KUKA KRL program: Station400_IMM.src, Station400_IMM.dat

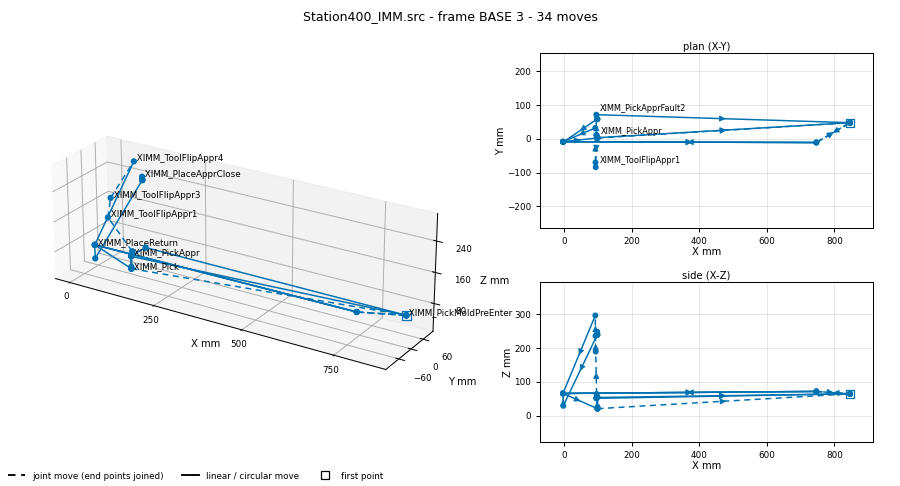
[picture p0: tool path of Station400_IMM.src in frame BASE 3, 34 of 42 moves have a stored position in this frame; points joined in program order, loops and branches not executed]
--- Station400_IMM.src ---
&ACCESS RVO1
&REL 170
&PARAM DISKPATH = KRC:\R1\Program
DEF Station400_IMM()
   ;FOLD INI;%{PE}
      ;FOLD BASISTECH INI
         GLOBAL INTERRUPT DECL 3 WHEN $STOPMESS == TRUE DO IR_STOPM()
         INTERRUPT ON 3
         BAS(#INITMOV, 0)
      ;ENDFOLD (BASISTECH INI)
      ;FOLD USER INI
         ;Make your modifications here
      ;ENDFOLD (USER INI)
      ;ENDFOLD (INI)
 RetryEntry:
 RtoIMM_MoldOpenEnable=True
 RtoPLC_FinishGripClose=False
 RtoPLC_FinishGripOpen=True
 wait sec .25
 RtoPLC_FinishGripOpen=False
 RobotCell_Error=False


;FOLD SPTP IMM_A1turn Vel=100 % PDAT4 Tool[0] Base[0] ;%{PE}
;FOLD Parameters ;%{h}
;Params IlfProvider=kukaroboter.basistech.inlineforms.movement.spline; Kuka.IsGlobalPoint=False; Kuka.PointName=IMM_A1turn; Kuka.BlendingEnabled=False; Kuka.MoveDataPtpName=PDAT4; Kuka.VelocityPtp=100; Kuka.VelocityFieldEnabled=True; Kuka.ColDetectFieldEnabled=True; Kuka.CurrentCDSetIndex=0; Kuka.MovementParameterFieldEnabled=True; IlfCommand=SPTP
;ENDFOLD
SPTP XIMM_A1turn WITH $VEL_AXIS[1] = SVEL_JOINT(100.0), $TOOL = STOOL2(FIMM_A1turn), $BASE = SBASE(FIMM_A1turn.BASE_NO), $IPO_MODE = SIPO_MODE(FIMM_A1turn.IPO_FRAME), $LOAD = SLOAD(FIMM_A1turn.TOOL_NO), $ACC_AXIS[1] = SACC_JOINT(PPDAT4), $APO = SAPO_PTP(PPDAT4), $GEAR_JERK[1] = SGEAR_JERK(PPDAT4), $COLLMON_TOL_PRO[1] = USE_CM_PRO_VALUES(0)
;ENDFOLD

Wait For IMMtoR_OpEnable==True
 Wait For RtoIMM_RobotWithIMM==False


;FOLD Wait for ejector backward signals,
$TIMER_STOP[2]=True ;stop timer
$TIMER[2]=0 ;reset timer
$TIMER_STOP[2]=False ;stop timer
Loop
       If $TIMER[2]>=5000 Then
              $TIMER_STOP[2]=True ;stop timer
              $TIMER[2]=0 ;reset timer
              IMMtoR_PreEntrErrorEjBck=True
              wait sec 0.25
              IMMtoR_PreEntrErrorEjBck=False
              Wait For IMMtoR_OpEnable==False
              GOTO RetryEntry
       EndIf
       If IMMtoR_EjectPosBck==True Then
              Exit
       EndIf
EndLoop
 ;ENDFOLD

;FOLD Wait for mold open signal, fault after 10 seconds of waiting, then move in over sprue, down and into mold pick position, turn on suction cups
$TIMER_STOP[2]=True ;stop timer
$TIMER[2]=0 ;reset timer
$TIMER_STOP[2]=False ;stop timer

Loop

       If $TIMER[2]>=5000 Then
              $TIMER_STOP[2]=True ;stop timer
              $TIMER[2]=0 ;reset timer
              IMMtoR_PlaceErrorMoldOpn=True
              wait sec 0.5
              IMMtoR_PlaceErrorMoldOpn=False
              Wait For IMMtoR_OpEnable==False
              GOTO RetryEntry
       EndIF

       If ((IMMtoR_MoldOpen==True) AND ((IMMtoR_PartInjected==True) Or (RtoIMM_SeqNumber<>0)))  Then
              If IMMtoR_Rejected==True Then
                     RtoPLC_ToolFinReject=True
              EndIf
              RtoIMM_MoldCloseEnable=False
              RtoIMM_MoldAreaFree=False
   ;FOLD SPTP IMM_PickMoldPreEnter CONT Vel=100 % PDAT1 Tool[2]:FinishedPlace Base[3]:IMM ;%{PE}
      ;FOLD Parameters ;%{h}
         ;Params IlfProvider=kukaroboter.basistech.inlineforms.movement.spline; Kuka.IsGlobalPoint=False; Kuka.PointName=IMM_PickMoldPreEnter; Kuka.BlendingEnabled=True; Kuka.MoveDataPtpName=PDAT1; Kuka.VelocityPtp=100; Kuka.VelocityFieldEnabled=True; Kuka.ColDetectFieldEnabled=True; Kuka.CurrentCDSetIndex=0; Kuka.MovementParameterFieldEnabled=True; IlfCommand=SPTP
      ;ENDFOLD
      SPTP XIMM_PickMoldPreEnter WITH $VEL_AXIS[1] = SVEL_JOINT(100.0), $TOOL = STOOL2(FIMM_PickMoldPreEnter), $BASE = SBASE(FIMM_PickMoldPreEnter.BASE_NO), $IPO_MODE = SIPO_MODE(FIMM_PickMoldPreEnter.IPO_FRAME), $LOAD = SLOAD(FIMM_PickMoldPreEnter.TOOL_NO), $ACC_AXIS[1] = SACC_JOINT(PPDAT1), $APO = SAPO_PTP(PPDAT1), $GEAR_JERK[1] = SGEAR_JERK(PPDAT1), $COLLMON_TOL_PRO[1] = USE_CM_PRO_VALUES(0) C_Spl
      ;ENDFOLD
;FOLD SLIN IMM_PickApprOvrSpru CONT Vel=1.5 m/s CPDAT01 Tool[1]:BlankPick Base[4]:SprueCutter ;%{PE}
;FOLD Parameters ;%{h}
;Params IlfProvider=kukaroboter.basistech.inlineforms.movement.spline; Kuka.IsGlobalPoint=False; Kuka.PointName=IMM_PickApprOvrSpru; Kuka.BlendingEnabled=True; Kuka.MoveDataName=CPDAT01; Kuka.VelocityPath=1.5; Kuka.VelocityFieldEnabled=True; Kuka.ColDetectFieldEnabled=True; Kuka.CurrentCDSetIndex=0; Kuka.MovementParameterFieldEnabled=True; IlfCommand=SLIN
;ENDFOLD
SLIN XIMM_PickApprOvrSpru WITH $VEL = SVEL_CP(1.5, , LCPDAT01), $TOOL = STOOL2(FIMM_PickApprOvrSpru), $BASE = SBASE(FIMM_PickApprOvrSpru.BASE_NO), $IPO_MODE = SIPO_MODE(FIMM_PickApprOvrSpru.IPO_FRAME), $LOAD = SLOAD(FIMM_PickApprOvrSpru.TOOL_NO), $ACC = SACC_CP(LCPDAT01), $ORI_TYPE = SORI_TYP(LCPDAT01), $APO = SAPO(LCPDAT01), $JERK = SJERK(LCPDAT01), $COLLMON_TOL_PRO[1] = USE_CM_PRO_VALUES(0) C_Spl
;ENDFOLD
;FOLD SLIN IMM_PickAppr Vel=1 m/s CPDAT2 Tool[2]:FinishedPlace Base[3]:IMM ;%{PE}
;FOLD Parameters ;%{h}
;Params IlfProvider=kukaroboter.basistech.inlineforms.movement.spline; Kuka.IsGlobalPoint=False; Kuka.PointName=IMM_PickAppr; Kuka.BlendingEnabled=False; Kuka.MoveDataName=CPDAT2; Kuka.VelocityPath=1; Kuka.VelocityFieldEnabled=True; Kuka.ColDetectFieldEnabled=True; Kuka.CurrentCDSetIndex=0; Kuka.MovementParameterFieldEnabled=True; IlfCommand=SLIN
;ENDFOLD
SLIN XIMM_PickAppr WITH $VEL = SVEL_CP(1.0, , LCPDAT2), $TOOL = STOOL2(FIMM_PickAppr), $BASE = SBASE(FIMM_PickAppr.BASE_NO), $IPO_MODE = SIPO_MODE(FIMM_PickAppr.IPO_FRAME), $LOAD = SLOAD(FIMM_PickAppr.TOOL_NO), $ACC = SACC_CP(LCPDAT2), $ORI_TYPE = SORI_TYP(LCPDAT2), $APO = SAPO(LCPDAT2), $JERK = SJERK(LCPDAT2), $COLLMON_TOL_PRO[1] = USE_CM_PRO_VALUES(0)
;ENDFOLD
;FOLD SLIN IMM_Pick Vel=0.05 m/s CPDAT1 Tool[2]:FinishedPlace Base[3]:IMM ;%{PE}
;FOLD Parameters ;%{h}
;Params IlfProvider=kukaroboter.basistech.inlineforms.movement.spline; Kuka.IsGlobalPoint=False; Kuka.PointName=IMM_Pick; Kuka.BlendingEnabled=False; Kuka.MoveDataName=CPDAT1; Kuka.VelocityPath=0.05; Kuka.VelocityFieldEnabled=True; Kuka.ColDetectFieldEnabled=True; Kuka.CurrentCDSetIndex=0; Kuka.MovementParameterFieldEnabled=True; IlfCommand=SLIN
;ENDFOLD
SLIN XIMM_Pick WITH $VEL = SVEL_CP(0.05, , LCPDAT1), $TOOL = STOOL2(FIMM_Pick), $BASE = SBASE(FIMM_Pick.BASE_NO), $IPO_MODE = SIPO_MODE(FIMM_Pick.IPO_FRAME), $LOAD = SLOAD(FIMM_Pick.TOOL_NO), $ACC = SACC_CP(LCPDAT1), $ORI_TYPE = SORI_TYP(LCPDAT1), $APO = SAPO(LCPDAT1), $JERK = SJERK(LCPDAT1), $COLLMON_TOL_PRO[1] = USE_CM_PRO_VALUES(0)
;ENDFOLD
              RtoPLC_FinishCupAVac=True
              RtoPLC_FinishCupBVac=True
              $TIMER_STOP[2]=True ;stop timer
              $TIMER[2]=0 ;reset timer
              Exit
       EndIf

       If ((IMMtoR_MoldOpen==True) AND ((IMMtoR_PartInjected==False) And (RtoIMM_SeqNumber==0)))  Then
              RtoIMM_MoldCloseEnable=False
              RtoIMM_MoldAreaFree=False
   ;FOLD SPTP IMM_PickMoldPreEnter CONT Vel=100 % PDAT1 Tool[2]:FinishedPlace Base[3]:IMM ;%{PE}
      ;FOLD Parameters ;%{h}
         ;Params IlfProvider=kukaroboter.basistech.inlineforms.movement.spline; Kuka.IsGlobalPoint=False; Kuka.PointName=IMM_PickMoldPreEnter; Kuka.BlendingEnabled=True; Kuka.MoveDataPtpName=PDAT1; Kuka.VelocityPtp=100; Kuka.VelocityFieldEnabled=True; Kuka.ColDetectFieldEnabled=True; Kuka.CurrentCDSetIndex=0; Kuka.MovementParameterFieldEnabled=True; IlfCommand=SPTP
      ;ENDFOLD
      SPTP XIMM_PickMoldPreEnter WITH $VEL_AXIS[1] = SVEL_JOINT(100.0), $TOOL = STOOL2(FIMM_PickMoldPreEnter), $BASE = SBASE(FIMM_PickMoldPreEnter.BASE_NO), $IPO_MODE = SIPO_MODE(FIMM_PickMoldPreEnter.IPO_FRAME), $LOAD = SLOAD(FIMM_PickMoldPreEnter.TOOL_NO), $ACC_AXIS[1] = SACC_JOINT(PPDAT1), $APO = SAPO_PTP(PPDAT1), $GEAR_JERK[1] = SGEAR_JERK(PPDAT1), $COLLMON_TOL_PRO[1] = USE_CM_PRO_VALUES(0) C_Spl
      ;ENDFOLD
;FOLD SPTP IMM_PlaceMoldReturn Vel=100 % PDAT15 Tool[1]:BlankPick Base[3]:IMM ;%{PE}
;FOLD Parameters ;%{h}
;Params IlfProvider=kukaroboter.basistech.inlineforms.movement.spline; Kuka.IsGlobalPoint=False; Kuka.PointName=IMM_PlaceMoldReturn; Kuka.BlendingEnabled=False; Kuka.MoveDataPtpName=PDAT15; Kuka.VelocityPtp=100; Kuka.VelocityFieldEnabled=True; Kuka.ColDetectFieldEnabled=True; Kuka.CurrentCDSetIndex=0; Kuka.MovementParameterFieldEnabled=True; IlfCommand=SPTP
;ENDFOLD
SPTP XIMM_PlaceMoldReturn WITH $VEL_AXIS[1] = SVEL_JOINT(100.0), $TOOL = STOOL2(FIMM_PlaceMoldReturn), $BASE = SBASE(FIMM_PlaceMoldReturn.BASE_NO), $IPO_MODE = SIPO_MODE(FIMM_PlaceMoldReturn.IPO_FRAME), $LOAD = SLOAD(FIMM_PlaceMoldReturn.TOOL_NO), $ACC_AXIS[1] = SACC_JOINT(PPDAT15), $APO = SAPO_PTP(PPDAT15), $GEAR_JERK[1] = SGEAR_JERK(PPDAT15), $COLLMON_TOL_PRO[1] = USE_CM_PRO_VALUES(0)
;ENDFOLD

;FOLD SLIN IMM_PlaceReturn Vel=2 m/s CPDAT23 Tool[1]:BlankPick Base[3]:IMM ;%{PE}
;FOLD Parameters ;%{h}
;Params IlfProvider=kukaroboter.basistech.inlineforms.movement.spline; Kuka.IsGlobalPoint=False; Kuka.PointName=IMM_PlaceReturn; Kuka.BlendingEnabled=False; Kuka.MoveDataName=CPDAT23; Kuka.VelocityPath=2; Kuka.VelocityFieldEnabled=True; Kuka.ColDetectFieldEnabled=True; Kuka.CurrentCDSetIndex=0; Kuka.MovementParameterFieldEnabled=True; IlfCommand=SLIN
;ENDFOLD
SLIN XIMM_PlaceReturn WITH $VEL = SVEL_CP(2.0, , LCPDAT23), $TOOL = STOOL2(FIMM_PlaceReturn), $BASE = SBASE(FIMM_PlaceReturn.BASE_NO), $IPO_MODE = SIPO_MODE(FIMM_PlaceReturn.IPO_FRAME), $LOAD = SLOAD(FIMM_PlaceReturn.TOOL_NO), $ACC = SACC_CP(LCPDAT23), $ORI_TYPE = SORI_TYP(LCPDAT23), $APO = SAPO(LCPDAT23), $JERK = SJERK(LCPDAT23), $COLLMON_TOL_PRO[1] = USE_CM_PRO_VALUES(0)
;ENDFOLD
              $TIMER_STOP[2]=True ;stop timer
              $TIMER[2]=0 ;reset timer
              GoTo PlaceInMold
       EndIf
EndLoop
;ENDFOLD

;FOLD Wait for suction cup vacuum signals, fault after 10 seconds of waiting (and back out of mold), move ejector forward,
$TIMER_STOP[2]=True ;stop timer
$TIMER[2]=0 ;reset timer
$TIMER_STOP[2]=False ;stop timer
Loop

       If $TIMER[2]>=5000 Then
              $TIMER_STOP[2]=True ;stop timer
              $TIMER[2]=0 ;reset timer
              If PLCtoR_FinishCupAVacOn==False Then
                     RtoIMM_PickErrorVG528=True

              EndIf
              If PLCtoR_FinishCupBVacOn==False Then
                     RtoIMM_PickErrorVG530=True

              EndIf
              Wait Sec .15
              RtoPLC_FinishCupAVac=False
              RtoPLC_FinishCupBVac=False
              RtoPLC_FinishCupABlow=True
              RtoPLC_FinishCupBBlow=True
              Wait Sec .15
              RtoPLC_FinishCupABlow=False
              RtoPLC_FinishCupBBlow=False
              RtoIMM_PickErrorVG528=False
              RtoIMM_PickErrorVG530=False
              Wait For IMMtoR_OpEnable==False
              $OV_PRO=30
              ;FOLD SLIN IMM_Pick Vel=0.05 m/s CPDAT1 Tool[2]:FinishedPlace Base[3]:IMM ;%{PE}
;FOLD Parameters ;%{h}
;Params IlfProvider=kukaroboter.basistech.inlineforms.movement.spline; Kuka.IsGlobalPoint=False; Kuka.PointName=IMM_Pick; Kuka.BlendingEnabled=False; Kuka.MoveDataName=CPDAT1; Kuka.VelocityPath=0.05; Kuka.VelocityFieldEnabled=True; Kuka.ColDetectFieldEnabled=True; Kuka.CurrentCDSetIndex=0; Kuka.MovementParameterFieldEnabled=True; IlfCommand=SLIN
;ENDFOLD
SLIN XIMM_Pick WITH $VEL = SVEL_CP(0.05, , LCPDAT1), $TOOL = STOOL2(FIMM_Pick), $BASE = SBASE(FIMM_Pick.BASE_NO), $IPO_MODE = SIPO_MODE(FIMM_Pick.IPO_FRAME), $LOAD = SLOAD(FIMM_Pick.TOOL_NO), $ACC = SACC_CP(LCPDAT1), $ORI_TYPE = SORI_TYP(LCPDAT1), $APO = SAPO(LCPDAT1), $JERK = SJERK(LCPDAT1), $COLLMON_TOL_PRO[1] = USE_CM_PRO_VALUES(0)
;ENDFOLD
;FOLD SLIN IMM_PickAppr Vel=1 m/s CPDAT2 Tool[2]:FinishedPlace Base[3]:IMM ;%{PE}
;FOLD Parameters ;%{h}
;Params IlfProvider=kukaroboter.basistech.inlineforms.movement.spline; Kuka.IsGlobalPoint=False; Kuka.PointName=IMM_PickAppr; Kuka.BlendingEnabled=False; Kuka.MoveDataName=CPDAT2; Kuka.VelocityPath=1; Kuka.VelocityFieldEnabled=True; Kuka.ColDetectFieldEnabled=True; Kuka.CurrentCDSetIndex=0; Kuka.MovementParameterFieldEnabled=True; IlfCommand=SLIN
;ENDFOLD
SLIN XIMM_PickAppr WITH $VEL = SVEL_CP(1.0, , LCPDAT2), $TOOL = STOOL2(FIMM_PickAppr), $BASE = SBASE(FIMM_PickAppr.BASE_NO), $IPO_MODE = SIPO_MODE(FIMM_PickAppr.IPO_FRAME), $LOAD = SLOAD(FIMM_PickAppr.TOOL_NO), $ACC = SACC_CP(LCPDAT2), $ORI_TYPE = SORI_TYP(LCPDAT2), $APO = SAPO(LCPDAT2), $JERK = SJERK(LCPDAT2), $COLLMON_TOL_PRO[1] = USE_CM_PRO_VALUES(0)
;ENDFOLD
;FOLD SLIN IMM_PickApprOvrSpru CONT Vel=1.5 m/s CPDAT01 Tool[1]:BlankPick Base[4]:SprueCutter ;%{PE}
;FOLD Parameters ;%{h}
;Params IlfProvider=kukaroboter.basistech.inlineforms.movement.spline; Kuka.IsGlobalPoint=False; Kuka.PointName=IMM_PickApprOvrSpru; Kuka.BlendingEnabled=True; Kuka.MoveDataName=CPDAT01; Kuka.VelocityPath=1.5; Kuka.VelocityFieldEnabled=True; Kuka.ColDetectFieldEnabled=True; Kuka.CurrentCDSetIndex=0; Kuka.MovementParameterFieldEnabled=True; IlfCommand=SLIN
;ENDFOLD
SLIN XIMM_PickApprOvrSpru WITH $VEL = SVEL_CP(1.5, , LCPDAT01), $TOOL = STOOL2(FIMM_PickApprOvrSpru), $BASE = SBASE(FIMM_PickApprOvrSpru.BASE_NO), $IPO_MODE = SIPO_MODE(FIMM_PickApprOvrSpru.IPO_FRAME), $LOAD = SLOAD(FIMM_PickApprOvrSpru.TOOL_NO), $ACC = SACC_CP(LCPDAT01), $ORI_TYPE = SORI_TYP(LCPDAT01), $APO = SAPO(LCPDAT01), $JERK = SJERK(LCPDAT01), $COLLMON_TOL_PRO[1] = USE_CM_PRO_VALUES(0) C_Spl
;ENDFOLD
;FOLD SLIN IMM_PickMoldPreEnter Vel=2 m/s CPDAT29 Tool[2]:FinishedPlace Base[3]:IMM ;%{PE}
;FOLD Parameters ;%{h}
;Params IlfProvider=kukaroboter.basistech.inlineforms.movement.spline; Kuka.IsGlobalPoint=False; Kuka.PointName=IMM_PickMoldPreEnter; Kuka.BlendingEnabled=False; Kuka.MoveDataName=CPDAT29; Kuka.VelocityPath=2; Kuka.VelocityFieldEnabled=True; Kuka.ColDetectFieldEnabled=True; Kuka.CurrentCDSetIndex=0; Kuka.MovementParameterFieldEnabled=True; IlfCommand=SLIN
;ENDFOLD
SLIN XIMM_PickMoldPreEnter WITH $VEL = SVEL_CP(2.0, , LCPDAT29), $TOOL = STOOL2(FIMM_PickMoldPreEnter), $BASE = SBASE(FIMM_PickMoldPreEnter.BASE_NO), $IPO_MODE = SIPO_MODE(FIMM_PickMoldPreEnter.IPO_FRAME), $LOAD = SLOAD(FIMM_PickMoldPreEnter.TOOL_NO), $ACC = SACC_CP(LCPDAT29), $ORI_TYPE = SORI_TYP(LCPDAT29), $APO = SAPO(LCPDAT29), $JERK = SJERK(LCPDAT29), $COLLMON_TOL_PRO[1] = USE_CM_PRO_VALUES(0)
;ENDFOLD
;FOLD SPTP IMM_A1Return Vel=100 % PDAT5 Tool[0] Base[0] ;%{PE}
;FOLD Parameters ;%{h}
;Params IlfProvider=kukaroboter.basistech.inlineforms.movement.spline; Kuka.IsGlobalPoint=False; Kuka.PointName=IMM_A1Return; Kuka.BlendingEnabled=False; Kuka.MoveDataPtpName=PDAT5; Kuka.VelocityPtp=100; Kuka.VelocityFieldEnabled=True; Kuka.ColDetectFieldEnabled=True; Kuka.CurrentCDSetIndex=0; Kuka.MovementParameterFieldEnabled=True; IlfCommand=SPTP
;ENDFOLD
SPTP XIMM_A1Return WITH $VEL_AXIS[1] = SVEL_JOINT(100.0), $TOOL = STOOL2(FIMM_A1Return), $BASE = SBASE(FIMM_A1Return.BASE_NO), $IPO_MODE = SIPO_MODE(FIMM_A1Return.IPO_FRAME), $LOAD = SLOAD(FIMM_A1Return.TOOL_NO), $ACC_AXIS[1] = SACC_JOINT(PPDAT5), $APO = SAPO_PTP(PPDAT5), $GEAR_JERK[1] = SGEAR_JERK(PPDAT5), $COLLMON_TOL_PRO[1] = USE_CM_PRO_VALUES(0)
;ENDFOLD
RtoIMM_MoldAreaFree=True
              Rjct_1Blnk_2Fin_3Both=2
              Station500_Reject()
              RtoIMM_SeqNumber=0
              GOTO EndOfModule
       EndIf

       If ((PLCtoR_FinishCupAVacOn==True) And (PLCtoR_FinishCupBVacOn==True)) Then
              $TIMER_STOP[2]=True ;stop timer
              $TIMER[2]=0 ;reset timer
              RtoIMM_MoldEjectFrw=True

              Exit
       EndIf

EndLoop
;ENDFOLD

;FOLD Wait for ejector forward signals, fault after 10 seconds of waiting (and back out of mold), Lift away part and send ejector backward
$TIMER_STOP[2]=True ;stop timer
$TIMER[2]=0 ;reset timer
$TIMER_STOP[2]=False ;stop timer
Loop
       If $TIMER[2]>=5000 Then
              $TIMER_STOP[2]=True ;stop timer
              $TIMER[2]=0 ;reset timer
              IMMtoR_PlaceErrorEjFrw=True
              Wait Sec .15
              IMMtoR_PlaceErrorEjFrw=False
              RtoIMM_MoldEjectFrw=False
              RtoPLC_FinishCupAVac=False
              RtoPLC_FinishCupBVac=False
              RtoPLC_FinishCupABlow=True
              RtoPLC_FinishCupBBlow=True
              Wait Sec .15
              RtoPLC_FinishCupABlow=False
              RtoPLC_FinishCupBBlow=False
              Wait For IMMtoR_OpEnable==False
              $OV_PRO=30
              ;FOLD SLIN IMM_Pick Vel=0.05 m/s CPDAT1 Tool[2]:FinishedPlace Base[3]:IMM ;%{PE}
;FOLD Parameters ;%{h}
;Params IlfProvider=kukaroboter.basistech.inlineforms.movement.spline; Kuka.IsGlobalPoint=False; Kuka.PointName=IMM_Pick; Kuka.BlendingEnabled=False; Kuka.MoveDataName=CPDAT1; Kuka.VelocityPath=0.05; Kuka.VelocityFieldEnabled=True; Kuka.ColDetectFieldEnabled=True; Kuka.CurrentCDSetIndex=0; Kuka.MovementParameterFieldEnabled=True; IlfCommand=SLIN
;ENDFOLD
SLIN XIMM_Pick WITH $VEL = SVEL_CP(0.05, , LCPDAT1), $TOOL = STOOL2(FIMM_Pick), $BASE = SBASE(FIMM_Pick.BASE_NO), $IPO_MODE = SIPO_MODE(FIMM_Pick.IPO_FRAME), $LOAD = SLOAD(FIMM_Pick.TOOL_NO), $ACC = SACC_CP(LCPDAT1), $ORI_TYPE = SORI_TYP(LCPDAT1), $APO = SAPO(LCPDAT1), $JERK = SJERK(LCPDAT1), $COLLMON_TOL_PRO[1] = USE_CM_PRO_VALUES(0)
;ENDFOLD
;FOLD SLIN IMM_PickApprFault Vel=0.5 m/s CPDAT31 Tool[2]:FinishedPlace Base[3]:IMM ;%{PE}
;FOLD Parameters ;%{h}
;Params IlfProvider=kukaroboter.basistech.inlineforms.movement.spline; Kuka.IsGlobalPoint=False; Kuka.PointName=IMM_PickApprFault; Kuka.BlendingEnabled=False; Kuka.MoveDataName=CPDAT31; Kuka.VelocityPath=0.5; Kuka.VelocityFieldEnabled=True; Kuka.ColDetectFieldEnabled=True; Kuka.CurrentCDSetIndex=0; Kuka.MovementParameterFieldEnabled=True; IlfCommand=SLIN
;ENDFOLD
SLIN XIMM_PickApprFault WITH $VEL = SVEL_CP(0.5, , LCPDAT31), $TOOL = STOOL2(FIMM_PickApprFault), $BASE = SBASE(FIMM_PickApprFault.BASE_NO), $IPO_MODE = SIPO_MODE(FIMM_PickApprFault.IPO_FRAME), $LOAD = SLOAD(FIMM_PickApprFault.TOOL_NO), $ACC = SACC_CP(LCPDAT31), $ORI_TYPE = SORI_TYP(LCPDAT31), $APO = SAPO(LCPDAT31), $JERK = SJERK(LCPDAT31), $COLLMON_TOL_PRO[1] = USE_CM_PRO_VALUES(0)
;ENDFOLD
;FOLD SLIN IMM_PickApprFault2 Vel=0.5 m/s CPDAT32 Tool[2]:FinishedPlace Base[3]:IMM ;%{PE}
;FOLD Parameters ;%{h}
;Params IlfProvider=kukaroboter.basistech.inlineforms.movement.spline; Kuka.IsGlobalPoint=False; Kuka.PointName=IMM_PickApprFault2; Kuka.BlendingEnabled=False; Kuka.MoveDataName=CPDAT32; Kuka.VelocityPath=0.5; Kuka.VelocityFieldEnabled=True; Kuka.ColDetectFieldEnabled=True; Kuka.CurrentCDSetIndex=0; Kuka.MovementParameterFieldEnabled=True; IlfCommand=SLIN
;ENDFOLD
SLIN XIMM_PickApprFault2 WITH $VEL = SVEL_CP(0.5, , LCPDAT32), $TOOL = STOOL2(FIMM_PickApprFault2), $BASE = SBASE(FIMM_PickApprFault2.BASE_NO), $IPO_MODE = SIPO_MODE(FIMM_PickApprFault2.IPO_FRAME), $LOAD = SLOAD(FIMM_PickApprFault2.TOOL_NO), $ACC = SACC_CP(LCPDAT32), $ORI_TYPE = SORI_TYP(LCPDAT32), $APO = SAPO(LCPDAT32), $JERK = SJERK(LCPDAT32), $COLLMON_TOL_PRO[1] = USE_CM_PRO_VALUES(0)
;ENDFOLD
;FOLD SLIN IMM_PickMoldPreEnter Vel=2 m/s CPDAT29 Tool[2]:FinishedPlace Base[3]:IMM ;%{PE}
;FOLD Parameters ;%{h}
;Params IlfProvider=kukaroboter.basistech.inlineforms.movement.spline; Kuka.IsGlobalPoint=False; Kuka.PointName=IMM_PickMoldPreEnter; Kuka.BlendingEnabled=False; Kuka.MoveDataName=CPDAT29; Kuka.VelocityPath=2; Kuka.VelocityFieldEnabled=True; Kuka.ColDetectFieldEnabled=True; Kuka.CurrentCDSetIndex=0; Kuka.MovementParameterFieldEnabled=True; IlfCommand=SLIN
;ENDFOLD
SLIN XIMM_PickMoldPreEnter WITH $VEL = SVEL_CP(2.0, , LCPDAT29), $TOOL = STOOL2(FIMM_PickMoldPreEnter), $BASE = SBASE(FIMM_PickMoldPreEnter.BASE_NO), $IPO_MODE = SIPO_MODE(FIMM_PickMoldPreEnter.IPO_FRAME), $LOAD = SLOAD(FIMM_PickMoldPreEnter.TOOL_NO), $ACC = SACC_CP(LCPDAT29), $ORI_TYPE = SORI_TYP(LCPDAT29), $APO = SAPO(LCPDAT29), $JERK = SJERK(LCPDAT29), $COLLMON_TOL_PRO[1] = USE_CM_PRO_VALUES(0)
;ENDFOLD
;FOLD SPTP IMM_A1Return Vel=100 % PDAT5 Tool[0] Base[0] ;%{PE}
;FOLD Parameters ;%{h}
;Params IlfProvider=kukaroboter.basistech.inlineforms.movement.spline; Kuka.IsGlobalPoint=False; Kuka.PointName=IMM_A1Return; Kuka.BlendingEnabled=False; Kuka.MoveDataPtpName=PDAT5; Kuka.VelocityPtp=100; Kuka.VelocityFieldEnabled=True; Kuka.ColDetectFieldEnabled=True; Kuka.CurrentCDSetIndex=0; Kuka.MovementParameterFieldEnabled=True; IlfCommand=SPTP
;ENDFOLD
SPTP XIMM_A1Return WITH $VEL_AXIS[1] = SVEL_JOINT(100.0), $TOOL = STOOL2(FIMM_A1Return), $BASE = SBASE(FIMM_A1Return.BASE_NO), $IPO_MODE = SIPO_MODE(FIMM_A1Return.IPO_FRAME), $LOAD = SLOAD(FIMM_A1Return.TOOL_NO), $ACC_AXIS[1] = SACC_JOINT(PPDAT5), $APO = SAPO_PTP(PPDAT5), $GEAR_JERK[1] = SGEAR_JERK(PPDAT5), $COLLMON_TOL_PRO[1] = USE_CM_PRO_VALUES(0)
;ENDFOLD
RtoIMM_MoldAreaFree=True
              Rjct_1Blnk_2Fin_3Both=2
              Station500_Reject()
              RtoIMM_SeqNumber=0
              GOTO EndOfModule
       Endif
       If IMMtoR_EjectPosFrw==True Then

;FOLD SLIN IMM_PickReturn2 Vel=0.05 m/s CPDAT22 Tool[2]:FinishedPlace Base[3]:IMM ;%{PE}
;FOLD Parameters ;%{h}
;Params IlfProvider=kukaroboter.basistech.inlineforms.movement.spline; Kuka.IsGlobalPoint=False; Kuka.PointName=IMM_PickReturn2; Kuka.BlendingEnabled=False; Kuka.MoveDataName=CPDAT22; Kuka.VelocityPath=0.05; Kuka.VelocityFieldEnabled=True; Kuka.ColDetectFieldEnabled=True; Kuka.CurrentCDSetIndex=0; Kuka.MovementParameterFieldEnabled=True; IlfCommand=SLIN
;ENDFOLD
SLIN XIMM_PickReturn2 WITH $VEL = SVEL_CP(0.05, , LCPDAT22), $TOOL = STOOL2(FIMM_PickReturn2), $BASE = SBASE(FIMM_PickReturn2.BASE_NO), $IPO_MODE = SIPO_MODE(FIMM_PickReturn2.IPO_FRAME), $LOAD = SLOAD(FIMM_PickReturn2.TOOL_NO), $ACC = SACC_CP(LCPDAT22), $ORI_TYPE = SORI_TYP(LCPDAT22), $APO = SAPO(LCPDAT22), $JERK = SJERK(LCPDAT22), $COLLMON_TOL_PRO[1] = USE_CM_PRO_VALUES(0)
;ENDFOLD
              RtoPLC_FinishGripClose=True
              Wait Sec .15

              RtoIMM_MoldEjectFrw=False
              Wait Sec .15
              RtoIMM_MoldEjectBack=True
                  ;FOLD SLIN IMM_PickReturn Vel=0.2 m/s CPDAT6 Tool[2]:TOOL_DATA[2] Base[3]:BASE_DATA[3] ;%{PE}
      ;FOLD Parameters ;%{h}
         ;Params IlfProvider=kukaroboter.basistech.inlineforms.movement.spline; Kuka.IsGlobalPoint=False; Kuka.PointName=IMM_PickReturn; Kuka.BlendingEnabled=False; Kuka.MoveDataName=CPDAT6; Kuka.VelocityPath=0.2; Kuka.VelocityFieldEnabled=True; Kuka.ColDetectFieldEnabled=True; Kuka.CurrentCDSetIndex=0; Kuka.MovementParameterFieldEnabled=True; IlfCommand=SLIN; SimId=
      ;ENDFOLD
      SLIN XIMM_PickReturn WITH $VEL = SVEL_CP(0.2, , LCPDAT6), $TOOL = STOOL2(FIMM_PickReturn), $BASE = SBASE(FIMM_PickReturn.BASE_NO), $IPO_MODE = SIPO_MODE(FIMM_PickReturn.IPO_FRAME), $LOAD = SLOAD(FIMM_PickReturn.TOOL_NO), $ACC = SACC_CP(LCPDAT6), $ORI_TYPE = SORI_TYP(LCPDAT6), $APO = SAPO(LCPDAT6), $JERK = SJERK(LCPDAT6), $COLLMON_TOL_PRO[1] = USE_CM_PRO_VALUES(0)
      ;ENDFOLD

              RtoPLC_ToolFinHasParts=True
              RtoPLC_ToolFinSeqNumber=RtoIMM_SeqNumber
              RtoIMM_SeqNumber=0
Exit
      EndIf
EndLoop
      ;ENDFOLD



;FOLD Wait for ejector backward signals, fault after 10 seconds of waiting (and back out of mold), Lift away part and send ejector backward
$TIMER_STOP[2]=True ;stop timer
$TIMER[2]=0 ;reset timer
$TIMER_STOP[2]=False ;stop timer
Loop
       If $TIMER[2]>=5000 Then
              $TIMER_STOP[2]=True ;stop timer
              $TIMER[2]=0 ;reset timer
              IMMtoR_PlaceErrorEjBck=True
              RtoIMM_MoldEjectBack=False
              Exit
       EndIf

       If IMMtoR_EjectPosBck==True Then
              Exit
       EndIf
EndLoop
 ;ENDFOLD

;FOLD if parts are in blank side of tooling, fault after 10 seconds of waiting (and back out of mold), if no fault, flip inside of mold and place parts, backout,

If ((RtoPLC_ToolBlnkHasParts==False) Or (IMMtoR_PlaceErrorEjBck==True)) Then
       Wait Sec .15
      IMMtoR_PlaceErrorEjBck=False
;FOLD SLIN IMM_PickMoldPreEnter CONT Vel=2 m/s CPDAT03 Tool[2]:FinishedPlace Base[3]:IMM ;%{PE}
;FOLD Parameters ;%{h}
;Params IlfProvider=kukaroboter.basistech.inlineforms.movement.spline; Kuka.IsGlobalPoint=False; Kuka.PointName=IMM_PickMoldPreEnter; Kuka.BlendingEnabled=True; Kuka.MoveDataName=CPDAT03; Kuka.VelocityPath=2; Kuka.VelocityFieldEnabled=True; Kuka.ColDetectFieldEnabled=True; Kuka.CurrentCDSetIndex=0; Kuka.MovementParameterFieldEnabled=True; IlfCommand=SLIN
;ENDFOLD
SLIN XIMM_PickMoldPreEnter WITH $VEL = SVEL_CP(2.0, , LCPDAT03), $TOOL = STOOL2(FIMM_PickMoldPreEnter), $BASE = SBASE(FIMM_PickMoldPreEnter.BASE_NO), $IPO_MODE = SIPO_MODE(FIMM_PickMoldPreEnter.IPO_FRAME), $LOAD = SLOAD(FIMM_PickMoldPreEnter.TOOL_NO), $ACC = SACC_CP(LCPDAT03), $ORI_TYPE = SORI_TYP(LCPDAT03), $APO = SAPO(LCPDAT03), $JERK = SJERK(LCPDAT03), $COLLMON_TOL_PRO[1] = USE_CM_PRO_VALUES(0) C_Spl
;ENDFOLD
;FOLD SPTP IMM_A1Return Vel=100 % PDAT5 Tool[0] Base[0] ;%{PE}
;FOLD Parameters ;%{h}
;Params IlfProvider=kukaroboter.basistech.inlineforms.movement.spline; Kuka.IsGlobalPoint=False; Kuka.PointName=IMM_A1Return; Kuka.BlendingEnabled=False; Kuka.MoveDataPtpName=PDAT5; Kuka.VelocityPtp=100; Kuka.VelocityFieldEnabled=True; Kuka.ColDetectFieldEnabled=True; Kuka.CurrentCDSetIndex=0; Kuka.MovementParameterFieldEnabled=True; IlfCommand=SPTP
;ENDFOLD
SPTP XIMM_A1Return WITH $VEL_AXIS[1] = SVEL_JOINT(100.0), $TOOL = STOOL2(FIMM_A1Return), $BASE = SBASE(FIMM_A1Return.BASE_NO), $IPO_MODE = SIPO_MODE(FIMM_A1Return.IPO_FRAME), $LOAD = SLOAD(FIMM_A1Return.TOOL_NO), $ACC_AXIS[1] = SACC_JOINT(PPDAT5), $APO = SAPO_PTP(PPDAT5), $GEAR_JERK[1] = SGEAR_JERK(PPDAT5), $COLLMON_TOL_PRO[1] = USE_CM_PRO_VALUES(0)
;ENDFOLD
RtoIMM_MoldAreaFree=True
       RtoIMM_MoldAreaFree=True
       RtoIMM_MoldCloseEnable=True
       If RtoPLC_ToolFinReject==True Then
              Rjct_1Blnk_2Fin_3Both=2
              Station500_Reject()
              GOTO EndOfModule
       EndIf
       GOTO EndOfModule
EndIf

If RtoPLC_ToolBlnkHasParts==True Then

;FOLD SPTP IMM_ToolFlipAppr CONT Vel=100 % PDAT8 Tool[2]:FinishedPlace Base[3]:IMM ;%{PE}
;FOLD Parameters ;%{h}
;Params IlfProvider=kukaroboter.basistech.inlineforms.movement.spline; Kuka.IsGlobalPoint=False; Kuka.PointName=IMM_ToolFlipAppr; Kuka.BlendingEnabled=True; Kuka.MoveDataPtpName=PDAT8; Kuka.VelocityPtp=100; Kuka.VelocityFieldEnabled=True; Kuka.ColDetectFieldEnabled=True; Kuka.CurrentCDSetIndex=0; Kuka.MovementParameterFieldEnabled=True; IlfCommand=SPTP
;ENDFOLD
SPTP XIMM_ToolFlipAppr WITH $VEL_AXIS[1] = SVEL_JOINT(100.0), $TOOL = STOOL2(FIMM_ToolFlipAppr), $BASE = SBASE(FIMM_ToolFlipAppr.BASE_NO), $IPO_MODE = SIPO_MODE(FIMM_ToolFlipAppr.IPO_FRAME), $LOAD = SLOAD(FIMM_ToolFlipAppr.TOOL_NO), $ACC_AXIS[1] = SACC_JOINT(PPDAT8), $APO = SAPO_PTP(PPDAT8), $GEAR_JERK[1] = SGEAR_JERK(PPDAT8), $COLLMON_TOL_PRO[1] = USE_CM_PRO_VALUES(0) C_Spl
;ENDFOLD

;FOLD SPTP IMM_ToolFlipAppr1 CONT Vel=100 % PDAT13 Tool[2]:FinishedPlace Base[3]:IMM ;%{PE}
;FOLD Parameters ;%{h}
;Params IlfProvider=kukaroboter.basistech.inlineforms.movement.spline; Kuka.IsGlobalPoint=False; Kuka.PointName=IMM_ToolFlipAppr1; Kuka.BlendingEnabled=True; Kuka.MoveDataPtpName=PDAT13; Kuka.VelocityPtp=100; Kuka.VelocityFieldEnabled=True; Kuka.ColDetectFieldEnabled=True; Kuka.CurrentCDSetIndex=0; Kuka.MovementParameterFieldEnabled=True; IlfCommand=SPTP
;ENDFOLD
SPTP XIMM_ToolFlipAppr1 WITH $VEL_AXIS[1] = SVEL_JOINT(100.0), $TOOL = STOOL2(FIMM_ToolFlipAppr1), $BASE = SBASE(FIMM_ToolFlipAppr1.BASE_NO), $IPO_MODE = SIPO_MODE(FIMM_ToolFlipAppr1.IPO_FRAME), $LOAD = SLOAD(FIMM_ToolFlipAppr1.TOOL_NO), $ACC_AXIS[1] = SACC_JOINT(PPDAT13), $APO = SAPO_PTP(PPDAT13), $GEAR_JERK[1] = SGEAR_JERK(PPDAT13), $COLLMON_TOL_PRO[1] = USE_CM_PRO_VALUES(0) C_Spl
;ENDFOLD


;FOLD SPTP IMM_ToolFlipAppr3 CONT Vel=100 % PDAT12 Tool[2]:FinishedPlace Base[3]:IMM ;%{PE}
;FOLD Parameters ;%{h}
;Params IlfProvider=kukaroboter.basistech.inlineforms.movement.spline; Kuka.IsGlobalPoint=False; Kuka.PointName=IMM_ToolFlipAppr3; Kuka.BlendingEnabled=True; Kuka.MoveDataPtpName=PDAT12; Kuka.VelocityPtp=100; Kuka.VelocityFieldEnabled=True; Kuka.ColDetectFieldEnabled=True; Kuka.CurrentCDSetIndex=0; Kuka.MovementParameterFieldEnabled=True; IlfCommand=SPTP
;ENDFOLD
SPTP XIMM_ToolFlipAppr3 WITH $VEL_AXIS[1] = SVEL_JOINT(100.0), $TOOL = STOOL2(FIMM_ToolFlipAppr3), $BASE = SBASE(FIMM_ToolFlipAppr3.BASE_NO), $IPO_MODE = SIPO_MODE(FIMM_ToolFlipAppr3.IPO_FRAME), $LOAD = SLOAD(FIMM_ToolFlipAppr3.TOOL_NO), $ACC_AXIS[1] = SACC_JOINT(PPDAT12), $APO = SAPO_PTP(PPDAT12), $GEAR_JERK[1] = SGEAR_JERK(PPDAT12), $COLLMON_TOL_PRO[1] = USE_CM_PRO_VALUES(0) C_Spl
;ENDFOLD

;FOLD SPTP IMM_ToolFlipAppr4 CONT Vel=100 % PDAT11 Tool[2]:FinishedPlace Base[3]:IMM ;%{PE}
;FOLD Parameters ;%{h}
;Params IlfProvider=kukaroboter.basistech.inlineforms.movement.spline; Kuka.IsGlobalPoint=False; Kuka.PointName=IMM_ToolFlipAppr4; Kuka.BlendingEnabled=True; Kuka.MoveDataPtpName=PDAT11; Kuka.VelocityPtp=100; Kuka.VelocityFieldEnabled=True; Kuka.ColDetectFieldEnabled=True; Kuka.CurrentCDSetIndex=0; Kuka.MovementParameterFieldEnabled=True; IlfCommand=SPTP
;ENDFOLD
SPTP XIMM_ToolFlipAppr4 WITH $VEL_AXIS[1] = SVEL_JOINT(100.0), $TOOL = STOOL2(FIMM_ToolFlipAppr4), $BASE = SBASE(FIMM_ToolFlipAppr4.BASE_NO), $IPO_MODE = SIPO_MODE(FIMM_ToolFlipAppr4.IPO_FRAME), $LOAD = SLOAD(FIMM_ToolFlipAppr4.TOOL_NO), $ACC_AXIS[1] = SACC_JOINT(PPDAT11), $APO = SAPO_PTP(PPDAT11), $GEAR_JERK[1] = SGEAR_JERK(PPDAT11), $COLLMON_TOL_PRO[1] = USE_CM_PRO_VALUES(0) C_Spl
;ENDFOLD

;FOLD SLIN IMM_PlaceReturn Vel=2 m/s CPDAT24 Tool[1]:BlankPick Base[3]:IMM ;%{PE}
;FOLD Parameters ;%{h}
;Params IlfProvider=kukaroboter.basistech.inlineforms.movement.spline; Kuka.IsGlobalPoint=False; Kuka.PointName=IMM_PlaceReturn; Kuka.BlendingEnabled=False; Kuka.MoveDataName=CPDAT24; Kuka.VelocityPath=2; Kuka.VelocityFieldEnabled=True; Kuka.ColDetectFieldEnabled=True; Kuka.CurrentCDSetIndex=0; Kuka.MovementParameterFieldEnabled=True; IlfCommand=SLIN
;ENDFOLD
SLIN XIMM_PlaceReturn WITH $VEL = SVEL_CP(2.0, , LCPDAT24), $TOOL = STOOL2(FIMM_PlaceReturn), $BASE = SBASE(FIMM_PlaceReturn.BASE_NO), $IPO_MODE = SIPO_MODE(FIMM_PlaceReturn.IPO_FRAME), $LOAD = SLOAD(FIMM_PlaceReturn.TOOL_NO), $ACC = SACC_CP(LCPDAT24), $ORI_TYPE = SORI_TYP(LCPDAT24), $APO = SAPO(LCPDAT24), $JERK = SJERK(LCPDAT24), $COLLMON_TOL_PRO[1] = USE_CM_PRO_VALUES(0)
;ENDFOLD


EndIf

PlaceInMold:
$TIMER_STOP[2]=True ;stop timer
$TIMER[2]=0 ;reset timer
$TIMER_STOP[2]=False ;stop timer

Loop
       If $TIMER[2]>=5000 Then
              $TIMER_STOP[2]=True ;stop timer
              $TIMER[2]=0 ;reset timer

              If PLCtoR_BlankCupAVacOn==False Then
                     RtoIMM_PlaceErrorVG524=True

              EndIf
              If PLCtoR_BlankCupBVacOn==False Then
                     RtoIMM_PlaceErrorVG526=True

              EndIf
              Wait Sec .15
              RtoIMM_PlaceErrorVG524=False
              RtoIMM_PlaceErrorVG526=False
              Wait For IMMtoR_OpEnable==False
              $OV_PRO=30
;FOLD SLIN IMM_PlaceReturn Vel=2 m/s CPDAT8 Tool[1]:BlankPick Base[3]:IMM ;%{PE}
;FOLD Parameters ;%{h}
;Params IlfProvider=kukaroboter.basistech.inlineforms.movement.spline; Kuka.IsGlobalPoint=False; Kuka.PointName=IMM_PlaceReturn; Kuka.BlendingEnabled=False; Kuka.MoveDataName=CPDAT8; Kuka.VelocityPath=2; Kuka.VelocityFieldEnabled=True; Kuka.ColDetectFieldEnabled=True; Kuka.CurrentCDSetIndex=0; Kuka.MovementParameterFieldEnabled=True; IlfCommand=SLIN
;ENDFOLD
SLIN XIMM_PlaceReturn WITH $VEL = SVEL_CP(2.0, , LCPDAT8), $TOOL = STOOL2(FIMM_PlaceReturn), $BASE = SBASE(FIMM_PlaceReturn.BASE_NO), $IPO_MODE = SIPO_MODE(FIMM_PlaceReturn.IPO_FRAME), $LOAD = SLOAD(FIMM_PlaceReturn.TOOL_NO), $ACC = SACC_CP(LCPDAT8), $ORI_TYPE = SORI_TYP(LCPDAT8), $APO = SAPO(LCPDAT8), $JERK = SJERK(LCPDAT8), $COLLMON_TOL_PRO[1] = USE_CM_PRO_VALUES(0)
;ENDFOLD
   ;FOLD SLIN IMM_PlaceMoldReturn CONT Vel=2 m/s CPDAT5 Tool[1]:TOOL_DATA[1] Base[3]:BASE_DATA[3] ;%{PE}
      ;FOLD Parameters ;%{h}
         ;Params IlfProvider=kukaroboter.basistech.inlineforms.movement.spline; Kuka.IsGlobalPoint=False; Kuka.PointName=IMM_PlaceMoldReturn; Kuka.BlendingEnabled=True; Kuka.MoveDataName=CPDAT5; Kuka.VelocityPath=2; Kuka.VelocityFieldEnabled=True; Kuka.ColDetectFieldEnabled=True; Kuka.CurrentCDSetIndex=0; Kuka.MovementParameterFieldEnabled=True; IlfCommand=SLIN
      ;ENDFOLD
      SLIN XIMM_PlaceMoldReturn WITH $VEL = SVEL_CP(2.0, , LCPDAT5), $TOOL = STOOL2(FIMM_PlaceMoldReturn), $BASE = SBASE(FIMM_PlaceMoldReturn.BASE_NO), $IPO_MODE = SIPO_MODE(FIMM_PlaceMoldReturn.IPO_FRAME), $LOAD = SLOAD(FIMM_PlaceMoldReturn.TOOL_NO), $ACC = SACC_CP(LCPDAT5), $ORI_TYPE = SORI_TYP(LCPDAT5), $APO = SAPO(LCPDAT5), $JERK = SJERK(LCPDAT5), $COLLMON_TOL_PRO[1] = USE_CM_PRO_VALUES(0) C_Spl
      ;ENDFOLD
         ;FOLD SPTP IMM_PickMoldPreEnter CONT Vel=100 % PDAT1 Tool[2]:FinishedPlace Base[3]:IMM ;%{PE}
      ;FOLD Parameters ;%{h}
         ;Params IlfProvider=kukaroboter.basistech.inlineforms.movement.spline; Kuka.IsGlobalPoint=False; Kuka.PointName=IMM_PickMoldPreEnter; Kuka.BlendingEnabled=True; Kuka.MoveDataPtpName=PDAT1; Kuka.VelocityPtp=100; Kuka.VelocityFieldEnabled=True; Kuka.ColDetectFieldEnabled=True; Kuka.CurrentCDSetIndex=0; Kuka.MovementParameterFieldEnabled=True; IlfCommand=SPTP
      ;ENDFOLD
      SPTP XIMM_PickMoldPreEnter WITH $VEL_AXIS[1] = SVEL_JOINT(100.0), $TOOL = STOOL2(FIMM_PickMoldPreEnter), $BASE = SBASE(FIMM_PickMoldPreEnter.BASE_NO), $IPO_MODE = SIPO_MODE(FIMM_PickMoldPreEnter.IPO_FRAME), $LOAD = SLOAD(FIMM_PickMoldPreEnter.TOOL_NO), $ACC_AXIS[1] = SACC_JOINT(PPDAT1), $APO = SAPO_PTP(PPDAT1), $GEAR_JERK[1] = SGEAR_JERK(PPDAT1), $COLLMON_TOL_PRO[1] = USE_CM_PRO_VALUES(0) C_Spl
      ;ENDFOLD
;FOLD SPTP IMM_A1Return Vel=100 % PDAT5 Tool[0] Base[0] ;%{PE}
;FOLD Parameters ;%{h}
;Params IlfProvider=kukaroboter.basistech.inlineforms.movement.spline; Kuka.IsGlobalPoint=False; Kuka.PointName=IMM_A1Return; Kuka.BlendingEnabled=False; Kuka.MoveDataPtpName=PDAT5; Kuka.VelocityPtp=100; Kuka.VelocityFieldEnabled=True; Kuka.ColDetectFieldEnabled=True; Kuka.CurrentCDSetIndex=0; Kuka.MovementParameterFieldEnabled=True; IlfCommand=SPTP
;ENDFOLD
SPTP XIMM_A1Return WITH $VEL_AXIS[1] = SVEL_JOINT(100.0), $TOOL = STOOL2(FIMM_A1Return), $BASE = SBASE(FIMM_A1Return.BASE_NO), $IPO_MODE = SIPO_MODE(FIMM_A1Return.IPO_FRAME), $LOAD = SLOAD(FIMM_A1Return.TOOL_NO), $ACC_AXIS[1] = SACC_JOINT(PPDAT5), $APO = SAPO_PTP(PPDAT5), $GEAR_JERK[1] = SGEAR_JERK(PPDAT5), $COLLMON_TOL_PRO[1] = USE_CM_PRO_VALUES(0)
;ENDFOLD
RtoIMM_MoldAreaFree=True
              Rjct_1Blnk_2Fin_3Both=1
              If RtoPLC_ToolFinReject==True Then
                     Rjct_1Blnk_2Fin_3Both=3
              EndIf
              Station500_Reject()
              GOTO EndOfModule
       EndIf

       If ((PLCtoR_BlankCupAVacOn==True) And (PLCtoR_BlankCupBVacOn==True)) Then

;FOLD SLIN IMM_PlaceApprClose Vel=1 m/s CPDAT14 Tool[2]:FinishedPlace Base[3]:IMM ;%{PE}
;FOLD Parameters ;%{h}
;Params IlfProvider=kukaroboter.basistech.inlineforms.movement.spline; Kuka.IsGlobalPoint=False; Kuka.PointName=IMM_PlaceApprClose; Kuka.BlendingEnabled=False; Kuka.MoveDataName=CPDAT14; Kuka.VelocityPath=1; Kuka.VelocityFieldEnabled=True; Kuka.ColDetectFieldEnabled=True; Kuka.CurrentCDSetIndex=0; Kuka.MovementParameterFieldEnabled=True; IlfCommand=SLIN
;ENDFOLD
SLIN XIMM_PlaceApprClose WITH $VEL = SVEL_CP(1.0, , LCPDAT14), $TOOL = STOOL2(FIMM_PlaceApprClose), $BASE = SBASE(FIMM_PlaceApprClose.BASE_NO), $IPO_MODE = SIPO_MODE(FIMM_PlaceApprClose.IPO_FRAME), $LOAD = SLOAD(FIMM_PlaceApprClose.TOOL_NO), $ACC = SACC_CP(LCPDAT14), $ORI_TYPE = SORI_TYP(LCPDAT14), $APO = SAPO(LCPDAT14), $JERK = SJERK(LCPDAT14), $COLLMON_TOL_PRO[1] = USE_CM_PRO_VALUES(0)
;ENDFOLD
;FOLD SLIN IMM_PlaceApprClose3 Vel=0.1 m/s CPDAT15 Tool[2]:FinishedPlace Base[3]:IMM ;%{PE}
;FOLD Parameters ;%{h}
;Params IlfProvider=kukaroboter.basistech.inlineforms.movement.spline; Kuka.IsGlobalPoint=False; Kuka.PointName=IMM_PlaceApprClose3; Kuka.BlendingEnabled=False; Kuka.MoveDataName=CPDAT15; Kuka.VelocityPath=0.1; Kuka.VelocityFieldEnabled=True; Kuka.ColDetectFieldEnabled=True; Kuka.CurrentCDSetIndex=0; Kuka.MovementParameterFieldEnabled=True; IlfCommand=SLIN
;ENDFOLD
SLIN XIMM_PlaceApprClose3 WITH $VEL = SVEL_CP(0.1, , LCPDAT15), $TOOL = STOOL2(FIMM_PlaceApprClose3), $BASE = SBASE(FIMM_PlaceApprClose3.BASE_NO), $IPO_MODE = SIPO_MODE(FIMM_PlaceApprClose3.IPO_FRAME), $LOAD = SLOAD(FIMM_PlaceApprClose3.TOOL_NO), $ACC = SACC_CP(LCPDAT15), $ORI_TYPE = SORI_TYP(LCPDAT15), $APO = SAPO(LCPDAT15), $JERK = SJERK(LCPDAT15), $COLLMON_TOL_PRO[1] = USE_CM_PRO_VALUES(0)
;ENDFOLD
;FOLD SLIN IMM_PlaceApprPushUp Vel=0.1 m/s CPDAT16 Tool[2]:FinishedPlace Base[3]:IMM ;%{PE}
;FOLD Parameters ;%{h}
;Params IlfProvider=kukaroboter.basistech.inlineforms.movement.spline; Kuka.IsGlobalPoint=False; Kuka.PointName=IMM_PlaceApprPushUp; Kuka.BlendingEnabled=False; Kuka.MoveDataName=CPDAT16; Kuka.VelocityPath=0.1; Kuka.VelocityFieldEnabled=True; Kuka.ColDetectFieldEnabled=True; Kuka.CurrentCDSetIndex=0; Kuka.MovementParameterFieldEnabled=True; IlfCommand=SLIN
;ENDFOLD
SLIN XIMM_PlaceApprPushUp WITH $VEL = SVEL_CP(0.1, , LCPDAT16), $TOOL = STOOL2(FIMM_PlaceApprPushUp), $BASE = SBASE(FIMM_PlaceApprPushUp.BASE_NO), $IPO_MODE = SIPO_MODE(FIMM_PlaceApprPushUp.IPO_FRAME), $LOAD = SLOAD(FIMM_PlaceApprPushUp.TOOL_NO), $ACC = SACC_CP(LCPDAT16), $ORI_TYPE = SORI_TYP(LCPDAT16), $APO = SAPO(LCPDAT16), $JERK = SJERK(LCPDAT16), $COLLMON_TOL_PRO[1] = USE_CM_PRO_VALUES(0)
;ENDFOLD

;FOLD LIN IMM_PlaceSideShft1 Vel=2 m/s CPDAT18 Tool[2]:FinishedPlace Base[3]:IMM ;%{PE}
;FOLD Parameters ;%{h}
;Params IlfProvider=kukaroboter.basistech.inlineforms.movement.old; Kuka.IsGlobalPoint=False; Kuka.PointName=IMM_PlaceSideShft1; Kuka.BlendingEnabled=False; Kuka.MoveDataName=CPDAT18; Kuka.VelocityPath=2; Kuka.CurrentCDSetIndex=0; Kuka.MovementParameterFieldEnabled=True; IlfCommand=LIN
;ENDFOLD
$BWDSTART = FALSE
LDAT_ACT = LCPDAT18
FDAT_ACT = FIMM_PlaceSideShft1
BAS(#CP_PARAMS, 2.0)
SET_CD_PARAMS (0)
LIN XIMM_PlaceSideShft1
;ENDFOLD
;FOLD SLIN IMM_PlaceSideShft2 Vel=2 m/s CPDAT19 Tool[2]:FinishedPlace Base[3]:IMM ;%{PE}
;FOLD Parameters ;%{h}
;Params IlfProvider=kukaroboter.basistech.inlineforms.movement.spline; Kuka.IsGlobalPoint=False; Kuka.PointName=IMM_PlaceSideShft2; Kuka.BlendingEnabled=False; Kuka.MoveDataName=CPDAT19; Kuka.VelocityPath=2; Kuka.VelocityFieldEnabled=True; Kuka.ColDetectFieldEnabled=True; Kuka.CurrentCDSetIndex=0; Kuka.MovementParameterFieldEnabled=True; IlfCommand=SLIN
;ENDFOLD
SLIN XIMM_PlaceSideShft2 WITH $VEL = SVEL_CP(2.0, , LCPDAT19), $TOOL = STOOL2(FIMM_PlaceSideShft2), $BASE = SBASE(FIMM_PlaceSideShft2.BASE_NO), $IPO_MODE = SIPO_MODE(FIMM_PlaceSideShft2.IPO_FRAME), $LOAD = SLOAD(FIMM_PlaceSideShft2.TOOL_NO), $ACC = SACC_CP(LCPDAT19), $ORI_TYPE = SORI_TYP(LCPDAT19), $APO = SAPO(LCPDAT19), $JERK = SJERK(LCPDAT19), $COLLMON_TOL_PRO[1] = USE_CM_PRO_VALUES(0)
;ENDFOLD
;FOLD SLIN IMM_PlaceSideShft3 Vel=2 m/s CPDAT20 Tool[2]:FinishedPlace Base[3]:IMM ;%{PE}
;FOLD Parameters ;%{h}
;Params IlfProvider=kukaroboter.basistech.inlineforms.movement.spline; Kuka.IsGlobalPoint=False; Kuka.PointName=IMM_PlaceSideShft3; Kuka.BlendingEnabled=False; Kuka.MoveDataName=CPDAT20; Kuka.VelocityPath=2; Kuka.VelocityFieldEnabled=True; Kuka.ColDetectFieldEnabled=True; Kuka.CurrentCDSetIndex=0; Kuka.MovementParameterFieldEnabled=True; IlfCommand=SLIN
;ENDFOLD
SLIN XIMM_PlaceSideShft3 WITH $VEL = SVEL_CP(2.0, , LCPDAT20), $TOOL = STOOL2(FIMM_PlaceSideShft3), $BASE = SBASE(FIMM_PlaceSideShft3.BASE_NO), $IPO_MODE = SIPO_MODE(FIMM_PlaceSideShft3.IPO_FRAME), $LOAD = SLOAD(FIMM_PlaceSideShft3.TOOL_NO), $ACC = SACC_CP(LCPDAT20), $ORI_TYPE = SORI_TYP(LCPDAT20), $APO = SAPO(LCPDAT20), $JERK = SJERK(LCPDAT20), $COLLMON_TOL_PRO[1] = USE_CM_PRO_VALUES(0)
;ENDFOLD

              RtoPLC_BlankCupAVac=False
              RtoPLC_BlankCupBVac=False
              RtoPLC_BlankCupABlow=True
              RtoPLC_BlankCupBBlow=True
;FOLD SLIN IMM_Place Vel=0.05 m/s CPDAT17 Tool[1]:BlankPick Base[3]:IMM ;%{PE}
;FOLD Parameters ;%{h}
;Params IlfProvider=kukaroboter.basistech.inlineforms.movement.spline; Kuka.IsGlobalPoint=False; Kuka.PointName=IMM_Place; Kuka.BlendingEnabled=False; Kuka.MoveDataName=CPDAT17; Kuka.VelocityPath=0.05; Kuka.VelocityFieldEnabled=True; Kuka.ColDetectFieldEnabled=True; Kuka.CurrentCDSetIndex=0; Kuka.MovementParameterFieldEnabled=True; IlfCommand=SLIN
;ENDFOLD
SLIN XIMM_Place WITH $VEL = SVEL_CP(0.05, , LCPDAT17), $TOOL = STOOL2(FIMM_Place), $BASE = SBASE(FIMM_Place.BASE_NO), $IPO_MODE = SIPO_MODE(FIMM_Place.IPO_FRAME), $LOAD = SLOAD(FIMM_Place.TOOL_NO), $ACC = SACC_CP(LCPDAT17), $ORI_TYPE = SORI_TYP(LCPDAT17), $APO = SAPO(LCPDAT17), $JERK = SJERK(LCPDAT17), $COLLMON_TOL_PRO[1] = USE_CM_PRO_VALUES(0)
;ENDFOLD

              Wait Sec .15
              RtoPLC_BlankCupABlow=False
              RtoPLC_BlankCupBBlow=False
              RtoIMM_SeqNumber=RtoPLC_ToolBlnkSeqNumber
              RtoPLC_ToolBlnkMrked=False
              RtoPLC_ToolBlnkSeqNumber=0
              RtoPLC_ToolBlnkHasParts=False

;FOLD SLIN IMM_PlaceReturn Vel=2 m/s CPDAT8 Tool[1]:BlankPick Base[3]:IMM ;%{PE}
;FOLD Parameters ;%{h}
;Params IlfProvider=kukaroboter.basistech.inlineforms.movement.spline; Kuka.IsGlobalPoint=False; Kuka.PointName=IMM_PlaceReturn; Kuka.BlendingEnabled=False; Kuka.MoveDataName=CPDAT8; Kuka.VelocityPath=2; Kuka.VelocityFieldEnabled=True; Kuka.ColDetectFieldEnabled=True; Kuka.CurrentCDSetIndex=0; Kuka.MovementParameterFieldEnabled=True; IlfCommand=SLIN
;ENDFOLD
SLIN XIMM_PlaceReturn WITH $VEL = SVEL_CP(2.0, , LCPDAT8), $TOOL = STOOL2(FIMM_PlaceReturn), $BASE = SBASE(FIMM_PlaceReturn.BASE_NO), $IPO_MODE = SIPO_MODE(FIMM_PlaceReturn.IPO_FRAME), $LOAD = SLOAD(FIMM_PlaceReturn.TOOL_NO), $ACC = SACC_CP(LCPDAT8), $ORI_TYPE = SORI_TYP(LCPDAT8), $APO = SAPO(LCPDAT8), $JERK = SJERK(LCPDAT8), $COLLMON_TOL_PRO[1] = USE_CM_PRO_VALUES(0)
;ENDFOLD
   ;FOLD SLIN IMM_PlaceMoldReturn CONT Vel=2 m/s CPDAT5 Tool[1]:TOOL_DATA[1] Base[3]:BASE_DATA[3] ;%{PE}
      ;FOLD Parameters ;%{h}
         ;Params IlfProvider=kukaroboter.basistech.inlineforms.movement.spline; Kuka.IsGlobalPoint=False; Kuka.PointName=IMM_PlaceMoldReturn; Kuka.BlendingEnabled=True; Kuka.MoveDataName=CPDAT5; Kuka.VelocityPath=2; Kuka.VelocityFieldEnabled=True; Kuka.ColDetectFieldEnabled=True; Kuka.CurrentCDSetIndex=0; Kuka.MovementParameterFieldEnabled=True; IlfCommand=SLIN
      ;ENDFOLD
      SLIN XIMM_PlaceMoldReturn WITH $VEL = SVEL_CP(2.0, , LCPDAT5), $TOOL = STOOL2(FIMM_PlaceMoldReturn), $BASE = SBASE(FIMM_PlaceMoldReturn.BASE_NO), $IPO_MODE = SIPO_MODE(FIMM_PlaceMoldReturn.IPO_FRAME), $LOAD = SLOAD(FIMM_PlaceMoldReturn.TOOL_NO), $ACC = SACC_CP(LCPDAT5), $ORI_TYPE = SORI_TYP(LCPDAT5), $APO = SAPO(LCPDAT5), $JERK = SJERK(LCPDAT5), $COLLMON_TOL_PRO[1] = USE_CM_PRO_VALUES(0) C_Spl
      ;ENDFOLD
         ;FOLD SPTP IMM_PickMoldPreEnter CONT Vel=100 % PDAT1 Tool[2]:FinishedPlace Base[3]:IMM ;%{PE}
      ;FOLD Parameters ;%{h}
         ;Params IlfProvider=kukaroboter.basistech.inlineforms.movement.spline; Kuka.IsGlobalPoint=False; Kuka.PointName=IMM_PickMoldPreEnter; Kuka.BlendingEnabled=True; Kuka.MoveDataPtpName=PDAT1; Kuka.VelocityPtp=100; Kuka.VelocityFieldEnabled=True; Kuka.ColDetectFieldEnabled=True; Kuka.CurrentCDSetIndex=0; Kuka.MovementParameterFieldEnabled=True; IlfCommand=SPTP
      ;ENDFOLD
      SPTP XIMM_PickMoldPreEnter WITH $VEL_AXIS[1] = SVEL_JOINT(100.0), $TOOL = STOOL2(FIMM_PickMoldPreEnter), $BASE = SBASE(FIMM_PickMoldPreEnter.BASE_NO), $IPO_MODE = SIPO_MODE(FIMM_PickMoldPreEnter.IPO_FRAME), $LOAD = SLOAD(FIMM_PickMoldPreEnter.TOOL_NO), $ACC_AXIS[1] = SACC_JOINT(PPDAT1), $APO = SAPO_PTP(PPDAT1), $GEAR_JERK[1] = SGEAR_JERK(PPDAT1), $COLLMON_TOL_PRO[1] = USE_CM_PRO_VALUES(0) C_Spl
      ;ENDFOLD
;FOLD SPTP IMM_A1Return Vel=100 % PDAT5 Tool[0] Base[0] ;%{PE}
;FOLD Parameters ;%{h}
;Params IlfProvider=kukaroboter.basistech.inlineforms.movement.spline; Kuka.IsGlobalPoint=False; Kuka.PointName=IMM_A1Return; Kuka.BlendingEnabled=False; Kuka.MoveDataPtpName=PDAT5; Kuka.VelocityPtp=100; Kuka.VelocityFieldEnabled=True; Kuka.ColDetectFieldEnabled=True; Kuka.CurrentCDSetIndex=0; Kuka.MovementParameterFieldEnabled=True; IlfCommand=SPTP
;ENDFOLD
SPTP XIMM_A1Return WITH $VEL_AXIS[1] = SVEL_JOINT(100.0), $TOOL = STOOL2(FIMM_A1Return), $BASE = SBASE(FIMM_A1Return.BASE_NO), $IPO_MODE = SIPO_MODE(FIMM_A1Return.IPO_FRAME), $LOAD = SLOAD(FIMM_A1Return.TOOL_NO), $ACC_AXIS[1] = SACC_JOINT(PPDAT5), $APO = SAPO_PTP(PPDAT5), $GEAR_JERK[1] = SGEAR_JERK(PPDAT5), $COLLMON_TOL_PRO[1] = USE_CM_PRO_VALUES(0)
;ENDFOLD
              RtoIMM_MoldAreaFree=True

              RtoIMM_MoldCloseEnable=True
              Exit
       EndIf
EndLoop

If RtoPLC_ToolFinReject==True Then
         Rjct_1Blnk_2Fin_3Both=2
         Station500_Reject()
EndIf

;ENDFOLD
EndofModule:
END

--- Station400_IMM.dat ---
&ACCESS RVP1
&REL 171
&PARAM DISKPATH = KRC:\R1\Program
DEFDAT  STATION400_IMM
;FOLD EXTERNAL DECLARATIONS;%{PE}%MKUKATPBASIS,%CEXT,%VCOMMON,%P
;FOLD BASISTECH EXT;%{PE}%MKUKATPBASIS,%CEXT,%VEXT,%P
EXT  BAS (BAS_COMMAND  :IN,REAL  :IN )
DECL INT SUCCESS
;ENDFOLD (BASISTECH EXT)
;FOLD USER EXT;%{E}%MKUKATPUSER,%CEXT,%VEXT,%P
;Make your modifications here

;ENDFOLD (USER EXT)
;ENDFOLD (EXTERNAL DECLARATIONS)
DECL LDAT LCPDAT1={VEL 0.0500000,ACC 60.0000,APO_DIST 500.000,APO_FAC 50.0000,AXIS_VEL 100.000,AXIS_ACC 60.0000,ORI_TYP #VAR,CIRC_TYP #BASE,JERK_FAC 50.0000,GEAR_JERK 100.000,EXAX_IGN 0,CB {AUX_PT {ORI #CONSIDER,E1 #CONSIDER,E2 #CONSIDER,E3 #CONSIDER,E4 #CONSIDER,E5 #CONSIDER,E6 #CONSIDER},TARGET_PT {ORI #INTERPOLATE,E1 #INTERPOLATE,E2 #INTERPOLATE,E3 #INTERPOLATE,E4 #INTERPOLATE,E5 #INTERPOLATE,E6 #INTERPOLATE}}}
DECL E6POS XIMM_Pick={X 98.4950638,Y 2.55296063,Z 20.6778107,A -90.3063202,B -1.35644746,C -179.035446,S 2,T 35,E1 0.0,E2 0.0,E3 0.0,E4 0.0,E5 0.0,E6 0.0}
DECL FDAT FIMM_Pick={TOOL_NO 2,BASE_NO 3,IPO_FRAME #BASE,POINT2[] " "}
DECL LDAT LCPDAT2={VEL 1.00000,ACC 60.0000,APO_DIST 500.000,APO_FAC 50.0000,AXIS_VEL 100.000,AXIS_ACC 60.0000,ORI_TYP #VAR,CIRC_TYP #BASE,JERK_FAC 50.0000,GEAR_JERK 100.000,EXAX_IGN 0,CB {AUX_PT {ORI #CONSIDER,E1 #CONSIDER,E2 #CONSIDER,E3 #CONSIDER,E4 #CONSIDER,E5 #CONSIDER,E6 #CONSIDER},TARGET_PT {ORI #INTERPOLATE,E1 #INTERPOLATE,E2 #INTERPOLATE,E3 #INTERPOLATE,E4 #INTERPOLATE,E5 #INTERPOLATE,E6 #INTERPOLATE}}}
DECL E6POS XIMM_PickAppr={X 97.9138260,Y 3.37952352,Z 55.4532127,A -90.3063202,B -1.35644746,C -179.035446,S 2,T 35,E1 0.0,E2 0.0,E3 0.0,E4 0.0,E5 0.0,E6 0.0}
DECL FDAT FIMM_PickAppr={TOOL_NO 2,BASE_NO 3,IPO_FRAME #BASE,POINT2[] " "}
DECL LDAT LCPDAT3={VEL 2.00000,ACC 60.0000,APO_DIST 500.000,APO_FAC 50.0000,AXIS_VEL 100.000,AXIS_ACC 60.0000,ORI_TYP #VAR,CIRC_TYP #BASE,JERK_FAC 50.0000,GEAR_JERK 100.000,EXAX_IGN 0}
DECL LDAT LCPDAT4={VEL 0.200000,ACC 60.0000,APO_DIST 500.000,APO_FAC 50.0000,AXIS_VEL 100.000,AXIS_ACC 60.0000,ORI_TYP #VAR,CIRC_TYP #BASE,JERK_FAC 50.0000,GEAR_JERK 100.000,EXAX_IGN 0}
DECL E6POS XIMM_Place={X -2.87502813,Y -9.41666889,Z 29.1462040,A 90.0059052,B 1.10676742,C -179.986374,S 2,T 35,E1 0.0,E2 0.0,E3 0.0,E4 0.0,E5 0.0,E6 0.0}
DECL FDAT FIMM_Place={TOOL_NO 1,BASE_NO 3,IPO_FRAME #BASE,POINT2[] " "}
DECL E6POS XIMM_PlaceAppr={X -6.11096096,Y -5.72452593,Z 58.3288460,A 90.0006638,B 2.66536307,C 179.556107,S 2,T 3,E1 0.0,E2 0.0,E3 0.0,E4 0.0,E5 0.0,E6 0.0}
DECL FDAT FIMM_PlaceAppr={TOOL_NO 1,BASE_NO 3,IPO_FRAME #BASE,POINT2[] " "}
DECL PDAT PDEFAULT={VEL 100.000,ACC 60.0000,APO_DIST 500.000,APO_MODE #CDIS,GEAR_JERK 100.000,EXAX_IGN 0}
DECL PDAT PPDAT1={VEL 100.000,ACC 60.0000,APO_DIST 500.000,APO_MODE #CDIS,GEAR_JERK 100.000,EXAX_IGN 0}
DECL PDAT PPDAT2={VEL 100.000,ACC 60.0000,APO_DIST 500.000,APO_MODE #CDIS,GEAR_JERK 100.000,EXAX_IGN 0}
DECL PDAT PPDAT3={VEL 100.000,ACC 60.0000,APO_DIST 500.000,APO_MODE #CDIS,GEAR_JERK 100.000,EXAX_IGN 0}
DECL PDAT PPDAT4={VEL 100.000,ACC 100.000,APO_DIST 500.000,APO_MODE #CDIS,GEAR_JERK 100.000,EXAX_IGN 0}
DECL LDAT LCPDAT5={VEL 2.00000,ACC 60.0000,APO_DIST 500.000,APO_FAC 50.0000,AXIS_VEL 100.000,AXIS_ACC 60.0000,ORI_TYP #VAR,CIRC_TYP #BASE,JERK_FAC 50.0000,GEAR_JERK 100.000,EXAX_IGN 0}
DECL PDAT PPDAT5={VEL 100.000,ACC 60.0000,APO_DIST 500.000,APO_MODE #CDIS,GEAR_JERK 100.000,EXAX_IGN 0}
DECL E6POS XIMM_A1turn={X -2.11590623E-11,Y 256.843719,Z 1087.90991,A -90.0000381,B 35.0000,C 179.999985,S 2,T 35,E1 0.0,E2 0.0,E3 0.0,E4 0.0,E5 0.0,E6 0.0}
DECL FDAT FIMM_A1turn={TOOL_NO 0,BASE_NO 0,IPO_FRAME #BASE,POINT2[] " "}
DECL LDAT LCPDAT6={VEL 2.00000,ACC 60.0000,APO_DIST 500.000,APO_FAC 50.0000,AXIS_VEL 100.000,AXIS_ACC 60.0000,ORI_TYP #VAR,CIRC_TYP #BASE,JERK_FAC 50.0000,GEAR_JERK 100.000,EXAX_IGN 0}
DECL PDAT PPDAT6={VEL 100.000,ACC 60.0000,APO_DIST 500.000,APO_MODE #CDIS,GEAR_JERK 100.000,EXAX_IGN 0}
DECL E6POS XIMM_ToolFlip={X 0.406555,Y -53.9616966,Z 57.8815918,A 90.2650299,B 1.36599696,C 179.049042,S 2,T 3,E1 0.0,E2 0.0,E3 0.0,E4 0.0,E5 0.0,E6 0.0}
DECL FDAT FIMM_ToolFlip={TOOL_NO 1,BASE_NO 3,IPO_FRAME #BASE,POINT2[] " "}
DECL LDAT LCPDAT7={VEL 0.200000,ACC 60.0000,APO_DIST 500.000,APO_FAC 50.0000,AXIS_VEL 100.000,AXIS_ACC 60.0000,ORI_TYP #VAR,CIRC_TYP #BASE,JERK_FAC 50.0000,GEAR_JERK 100.000,EXAX_IGN 0}
DECL E6POS XIMM_PickMoldPreEnter={X 846.035,Y 47.7981606,Z 64.6274109,A -90.3063202,B -1.35643947,C -179.035446,S 2,T 35,E1 0.0,E2 0.0,E3 0.0,E4 0.0,E5 0.0,E6 0.0}
DECL FDAT FIMM_PickMoldPreEnter={TOOL_NO 2,BASE_NO 3,IPO_FRAME #BASE,POINT2[] " "}
DECL E6POS XIMM_A1Return={X -1.04082927E-13,Y 256.843719,Z 1087.90991,A -90.0000381,B 35.0000,C 179.999985,S 2,T 35,E1 0.0,E2 0.0,E3 0.0,E4 0.0,E5 0.0,E6 0.0}
DECL FDAT FIMM_A1Return={TOOL_NO 0,BASE_NO 0,IPO_FRAME #BASE,POINT2[] " "}
DECL E6POS XIMM_PickReturn={X 97.9425201,Y 3.33871484,Z 53.7363358,A -90.3063202,B -1.35644746,C -179.035446,S 2,T 35,E1 0.0,E2 0.0,E3 0.0,E4 0.0,E5 0.0,E6 0.0}
DECL FDAT FIMM_PickReturn={TOOL_NO 2,BASE_NO 3,IPO_FRAME #BASE,POINT2[] " "}
DECL E6POS XIMM_PlaceReturn={X -3.77914834,Y -8.53857899,Z 65.7790,A 90.0057373,B 1.52101529,C 179.551056,S 2,T 35,E1 0.0,E2 0.0,E3 0.0,E4 0.0,E5 0.0,E6 0.0}
DECL FDAT FIMM_PlaceReturn={TOOL_NO 1,BASE_NO 3,IPO_FRAME #BASE,POINT2[] " "}
DECL E6POS XIMM_PlaceMoldReturn={X 746.193481,Y -10.9245615,Z 71.7229843,A 90.0057373,B 1.52101529,C 179.551056,S 2,T 35,E1 0.0,E2 0.0,E3 0.0,E4 0.0,E5 0.0,E6 0.0}
DECL FDAT FIMM_PlaceMoldReturn={TOOL_NO 1,BASE_NO 3,IPO_FRAME #BASE,POINT2[] " "}
DECL E6POS XIMM_PickApprOvrSpru={X 824.909485,Y 461.549774,Z 1451.45325,A -89.4070,B -0.628342271,C -90.0015,S 2,T 35,E1 0.0,E2 0.0,E3 0.0,E4 0.0,E5 0.0,E6 0.0}
DECL FDAT FIMM_PickApprOvrSpru={TOOL_NO 1,BASE_NO 4,IPO_FRAME #BASE,POINT2[] " "}
DECL LDAT LCPDAT01={VEL 1.50000,ACC 60.0000,APO_DIST 100.000,APO_FAC 50.0000,AXIS_VEL 100.000,AXIS_ACC 60.0000,ORI_TYP #VAR,CIRC_TYP #BASE,JERK_FAC 50.0000,GEAR_JERK 100.000,EXAX_IGN 0,CB {AUX_PT {ORI #CONSIDER,E1 #CONSIDER,E2 #CONSIDER,E3 #CONSIDER,E4 #CONSIDER,E5 #CONSIDER,E6 #CONSIDER},TARGET_PT {ORI #INTERPOLATE,E1 #INTERPOLATE,E2 #INTERPOLATE,E3 #INTERPOLATE,E4 #INTERPOLATE,E5 #INTERPOLATE,E6 #INTERPOLATE}}}
DECL MODULEPARAM_T LAST_TP_PARAMS={PARAMS[] "Kuka.VelocityFieldEnabled=True; Kuka.ColDetectFieldEnabled=True; Kuka.MovementParameterFieldEnabled=True; Kuka.IsAngleEnabled=False; Kuka.PointName=IMM_PickApprOvrSpru; Kuka.FrameData.base_no=4; Kuka.FrameData.tool_no=1; Kuka.FrameData.ipo_frame=#BASE; Kuka.FrameData.point2=; Kuka.isglobalpoint=False; Kuka.MoveDataName=CPDAT01; Kuka.MovementData.cb={AUX_PT {ORI #CONSIDER,E1 #CONSIDER,E2 #CONSIDER,E3 #CONSIDER,E4 #CONSIDER,E5 #CONSIDER,E6 #CONSIDER},TARGET_PT {ORI #INTERPOLATE,E1 #INTERPOLATE,E2 #INTERPOLATE,E3 #INTERPOLATE,E4 #INTERPOLATE,E5 #INTERPOLATE,E6 #INTERPOLATE}}; Kuka.MovementData.apo_fac=50; Kuka.MovementData.apo_dist=100; Kuka.MovementData.axis_acc=60; Kuka.MovementData.axis_vel=100; Kuka.MovementData.circ_typ=#BASE; Kuka.MovementData.jerk_fac=50; Kuka.MovementData.ori_typ=#VAR; Kuka.MovementData.vel=1.5; Kuka.MovementData.acc=60; Kuka.MovementData.exax_ign=0; Kuka.VelocityPath=1.5; Kuka.BlendingEnabled=True; Kuka.APXEnabled=False; Kuka.CurrentCDSetIndex=0; Kuka.MoveDataPtpName=PDAT4; Kuka.MovementDataPdat.apo_mode=#CDIS; Kuka.MovementDataPdat.apo_dist=500; Kuka.VelocityPtp=100      "}
DECL LDAT LCPDAT02={VEL 2.00000,ACC 60.0000,APO_DIST 500.000,APO_FAC 50.0000,AXIS_VEL 100.000,AXIS_ACC 60.0000,ORI_TYP #VAR,CIRC_TYP #BASE,JERK_FAC 50.0000,GEAR_JERK 100.000,EXAX_IGN 0,CB {AUX_PT {ORI #CONSIDER,E1 #CONSIDER,E2 #CONSIDER,E3 #CONSIDER,E4 #CONSIDER,E5 #CONSIDER,E6 #CONSIDER},TARGET_PT {ORI #INTERPOLATE,E1 #INTERPOLATE,E2 #INTERPOLATE,E3 #INTERPOLATE,E4 #INTERPOLATE,E5 #INTERPOLATE,E6 #INTERPOLATE}}}
DECL LDAT LCPDAT03={VEL 2.00000,ACC 60.0000,APO_DIST 500.000,APO_FAC 50.0000,AXIS_VEL 100.000,AXIS_ACC 60.0000,ORI_TYP #VAR,CIRC_TYP #BASE,JERK_FAC 50.0000,GEAR_JERK 100.000,EXAX_IGN 0,CB {AUX_PT {ORI #CONSIDER,E1 #CONSIDER,E2 #CONSIDER,E3 #CONSIDER,E4 #CONSIDER,E5 #CONSIDER,E6 #CONSIDER},TARGET_PT {ORI #INTERPOLATE,E1 #INTERPOLATE,E2 #INTERPOLATE,E3 #INTERPOLATE,E4 #INTERPOLATE,E5 #INTERPOLATE,E6 #INTERPOLATE}}}
DECL PDAT PPDAT7={VEL 100.000,ACC 60.0000,APO_DIST 500.000,APO_MODE #CDIS,GEAR_JERK 100.000,EXAX_IGN 0}
DECL FDAT FIMM_A1turn_1={TOOL_NO 0,BASE_NO 0,IPO_FRAME #BASE,POINT2[] " "}
DECL E6POS XIMM_A1turn_1={X -2.11590623E-11,Y 256.843719,Z 1087.90991,A -90.0000381,B 35.0000,C 179.999985,S 2,T 35,E1 0.0,E2 0.0,E3 0.0,E4 0.0,E5 0.0,E6 0.0}
DECL E6POS XIMM_PickMold1={X 666666.688,Y 66.6000,Z 666.660,A 6.60000,B 66.6600,C 666.600,S 0,T 0,E1 0.0,E2 0.0,E3 0.0,E4 0.0,E5 0.0,E6 0.0}
DECL FDAT FIMM_PickMold1={TOOL_NO 2,BASE_NO 3,IPO_FRAME #BASE,POINT2[] " "}
DECL LDAT LCPDAT04={VEL 0.100000,ACC 60.0000,APO_DIST 500.000,APO_FAC 50.0000,AXIS_VEL 100.000,AXIS_ACC 60.0000,ORI_TYP #VAR,CIRC_TYP #BASE,JERK_FAC 50.0000,GEAR_JERK 100.000,EXAX_IGN 0,CB {AUX_PT {ORI #CONSIDER,E1 #CONSIDER,E2 #CONSIDER,E3 #CONSIDER,E4 #CONSIDER,E5 #CONSIDER,E6 #CONSIDER},TARGET_PT {ORI #INTERPOLATE,E1 #INTERPOLATE,E2 #INTERPOLATE,E3 #INTERPOLATE,E4 #INTERPOLATE,E5 #INTERPOLATE,E6 #INTERPOLATE}}}
DECL E6POS XIMM_PickMold={X 666666.688,Y 66.6000,Z 666.660,A 6.60000,B 66.6600,C 666.600,S 0,T 0,E1 0.0,E2 0.0,E3 0.0,E4 0.0,E5 0.0,E6 0.0}
DECL FDAT FIMM_PickMold={TOOL_NO 2,BASE_NO 3,IPO_FRAME #BASE,POINT2[] " "}
DECL LDAT LCPDAT05={VEL 0.100000,ACC 60.0000,APO_DIST 500.000,APO_FAC 50.0000,AXIS_VEL 100.000,AXIS_ACC 60.0000,ORI_TYP #VAR,CIRC_TYP #BASE,JERK_FAC 50.0000,GEAR_JERK 100.000,EXAX_IGN 0,CB {AUX_PT {ORI #CONSIDER,E1 #CONSIDER,E2 #CONSIDER,E3 #CONSIDER,E4 #CONSIDER,E5 #CONSIDER,E6 #CONSIDER},TARGET_PT {ORI #INTERPOLATE,E1 #INTERPOLATE,E2 #INTERPOLATE,E3 #INTERPOLATE,E4 #INTERPOLATE,E5 #INTERPOLATE,E6 #INTERPOLATE}}}
DECL E6POS XIMM_PickReturn1={X 96.5922623,Y 10.1557093,Z 13.5926523,A -90.3063202,B -1.35644317,C -179.035446,S 2,T 35,E1 0.0,E2 0.0,E3 0.0,E4 0.0,E5 0.0,E6 0.0}
DECL FDAT FIMM_PickReturn1={TOOL_NO 2,BASE_NO 3,IPO_FRAME #BASE,POINT2[] " "}
DECL LDAT LCPDAT06={VEL 0.100000,ACC 60.0000,APO_DIST 500.000,APO_FAC 50.0000,AXIS_VEL 100.000,AXIS_ACC 60.0000,ORI_TYP #VAR,CIRC_TYP #BASE,JERK_FAC 50.0000,GEAR_JERK 100.000,EXAX_IGN 0,CB {AUX_PT {ORI #CONSIDER,E1 #CONSIDER,E2 #CONSIDER,E3 #CONSIDER,E4 #CONSIDER,E5 #CONSIDER,E6 #CONSIDER},TARGET_PT {ORI #INTERPOLATE,E1 #INTERPOLATE,E2 #INTERPOLATE,E3 #INTERPOLATE,E4 #INTERPOLATE,E5 #INTERPOLATE,E6 #INTERPOLATE}}}
DECL E6POS XIMM_PickReturn2={X 98.4073334,Y 2.67771554,Z 25.9265537,A -90.3063202,B -1.35644746,C -179.035446,S 2,T 35,E1 0.0,E2 0.0,E3 0.0,E4 0.0,E5 0.0,E6 0.0}
DECL FDAT FIMM_PickReturn2={TOOL_NO 2,BASE_NO 3,IPO_FRAME #BASE,POINT2[] " "}
DECL LDAT LCPDAT07={VEL 0.100000,ACC 60.0000,APO_DIST 500.000,APO_FAC 50.0000,AXIS_VEL 100.000,AXIS_ACC 60.0000,ORI_TYP #VAR,CIRC_TYP #BASE,JERK_FAC 50.0000,GEAR_JERK 100.000,EXAX_IGN 0,CB {AUX_PT {ORI #CONSIDER,E1 #CONSIDER,E2 #CONSIDER,E3 #CONSIDER,E4 #CONSIDER,E5 #CONSIDER,E6 #CONSIDER},TARGET_PT {ORI #INTERPOLATE,E1 #INTERPOLATE,E2 #INTERPOLATE,E3 #INTERPOLATE,E4 #INTERPOLATE,E5 #INTERPOLATE,E6 #INTERPOLATE}}}
DECL E6POS XIMM_ToolFlipAppr={X 95.7469482,Y 11.3577900,Z 64.1679535,A -90.3063202,B -1.35644329,C -179.035446,S 2,T 35,E1 0.0,E2 0.0,E3 0.0,E4 0.0,E5 0.0,E6 0.0}
DECL FDAT FIMM_ToolFlipAppr={TOOL_NO 2,BASE_NO 3,IPO_FRAME #BASE,POINT2[] " "}
DECL PDAT PPDAT8={VEL 100.000,ACC 60.0000,APO_DIST 500.000,APO_MODE #CDIS,GEAR_JERK 100.000,EXAX_IGN 0}
DECL E6POS XIMM_ToolFlipAppr1={X 93.1607361,Y -84.0203476,Z 189.797485,A 108.974976,B -87.0781479,C -19.2815018,S 2,T 35,E1 0.0,E2 0.0,E3 0.0,E4 0.0,E5 0.0,E6 0.0}
DECL FDAT FIMM_ToolFlipAppr1={TOOL_NO 2,BASE_NO 3,IPO_FRAME #BASE,POINT2[] " "}
DECL PDAT PPDAT9={VEL 100.000,ACC 60.0000,APO_DIST 500.000,APO_MODE #CDIS,GEAR_JERK 100.000,EXAX_IGN 0}
DECL LDAT LCPDAT08={VEL 0.100000,ACC 60.0000,APO_DIST 500.000,APO_FAC 50.0000,AXIS_VEL 100.000,AXIS_ACC 60.0000,ORI_TYP #VAR,CIRC_TYP #BASE,JERK_FAC 50.0000,GEAR_JERK 100.000,EXAX_IGN 0,CB {AUX_PT {ORI #CONSIDER,E1 #CONSIDER,E2 #CONSIDER,E3 #CONSIDER,E4 #CONSIDER,E5 #CONSIDER,E6 #CONSIDER},TARGET_PT {ORI #INTERPOLATE,E1 #INTERPOLATE,E2 #INTERPOLATE,E3 #INTERPOLATE,E4 #INTERPOLATE,E5 #INTERPOLATE,E6 #INTERPOLATE}}}
DECL E6POS XIMM_ToolFlipAppr2={X 92.6466141,Y -75.2470627,Z 222.919678,A 92.1252213,B -68.1692886,C -2.59428334,S 2,T 35,E1 0.0,E2 0.0,E3 0.0,E4 0.0,E5 0.0,E6 0.0}
DECL FDAT FIMM_ToolFlipAppr2={TOOL_NO 2,BASE_NO 3,IPO_FRAME #BASE,POINT2[] " "}
DECL PDAT PPDAT10={VEL 100.000,ACC 60.0000,APO_DIST 500.000,APO_MODE #CDIS,GEAR_JERK 100.000,EXAX_IGN 0}
DECL E6POS XIMM_ToolFlipAppr3={X 92.4512711,Y -69.9831085,Z 236.069122,A 92.1252213,B -68.1692886,C -2.59428334,S 2,T 35,E1 0.0,E2 0.0,E3 0.0,E4 0.0,E5 0.0,E6 0.0}
DECL FDAT FIMM_ToolFlipAppr3={TOOL_NO 2,BASE_NO 3,IPO_FRAME #BASE,POINT2[] " "}
DECL LDAT LCPDAT09={VEL 0.100000,ACC 60.0000,APO_DIST 500.000,APO_FAC 50.0000,AXIS_VEL 100.000,AXIS_ACC 60.0000,ORI_TYP #VAR,CIRC_TYP #BASE,JERK_FAC 50.0000,GEAR_JERK 100.000,EXAX_IGN 0,CB {AUX_PT {ORI #CONSIDER,E1 #CONSIDER,E2 #CONSIDER,E3 #CONSIDER,E4 #CONSIDER,E5 #CONSIDER,E6 #CONSIDER},TARGET_PT {ORI #INTERPOLATE,E1 #INTERPOLATE,E2 #INTERPOLATE,E3 #INTERPOLATE,E4 #INTERPOLATE,E5 #INTERPOLATE,E6 #INTERPOLATE}}}
DECL E6POS XIMM_ToolFlipAppr4={X 91.9377747,Y 32.2032051,Z 296.596863,A 89.6863632,B 1.81151450,C -0.964756310,S 2,T 35,E1 0.0,E2 0.0,E3 0.0,E4 0.0,E5 0.0,E6 0.0}
DECL FDAT FIMM_ToolFlipAppr4={TOOL_NO 2,BASE_NO 3,IPO_FRAME #BASE,POINT2[] " "}
DECL PDAT PPDAT11={VEL 100.000,ACC 60.0000,APO_DIST 500.000,APO_MODE #CDIS,GEAR_JERK 100.000,EXAX_IGN 0}
DECL E6POS XIMM_PlaceApprClose={X 97.6729736,Y 58.1790390,Z 248.257401,A 90.0060806,B 1.10676742,C 0.0136310831,S 2,T 35,E1 0.0,E2 0.0,E3 0.0,E4 0.0,E5 0.0,E6 0.0}
DECL FDAT FIMM_PlaceApprClose={TOOL_NO 2,BASE_NO 3,IPO_FRAME #BASE,POINT2[] " "}
DECL LDAT LCPDAT10={VEL 2.00000,ACC 60.0000,APO_DIST 500.000,APO_FAC 50.0000,AXIS_VEL 100.000,AXIS_ACC 60.0000,ORI_TYP #VAR,CIRC_TYP #BASE,JERK_FAC 50.0000,GEAR_JERK 100.000,EXAX_IGN 0,CB {AUX_PT {ORI #CONSIDER,E1 #CONSIDER,E2 #CONSIDER,E3 #CONSIDER,E4 #CONSIDER,E5 #CONSIDER,E6 #CONSIDER},TARGET_PT {ORI #INTERPOLATE,E1 #INTERPOLATE,E2 #INTERPOLATE,E3 #INTERPOLATE,E4 #INTERPOLATE,E5 #INTERPOLATE,E6 #INTERPOLATE}}}
DECL E6POS XIMM_PlaceApprClose2={X 93.2400513,Y 64.7528610,Z 231.462875,A 89.6777115,B 2.32530260,C -0.963273406,S 2,T 35,E1 0.0,E2 0.0,E3 0.0,E4 0.0,E5 0.0,E6 0.0}
DECL FDAT FIMM_PlaceApprClose2={TOOL_NO 2,BASE_NO 3,IPO_FRAME #BASE,POINT2[] " "}
DECL LDAT LCPDAT11={VEL 0.100000,ACC 60.0000,APO_DIST 500.000,APO_FAC 50.0000,AXIS_VEL 100.000,AXIS_ACC 60.0000,ORI_TYP #VAR,CIRC_TYP #BASE,JERK_FAC 50.0000,GEAR_JERK 100.000,EXAX_IGN 0,CB {AUX_PT {ORI #CONSIDER,E1 #CONSIDER,E2 #CONSIDER,E3 #CONSIDER,E4 #CONSIDER,E5 #CONSIDER,E6 #CONSIDER},TARGET_PT {ORI #INTERPOLATE,E1 #INTERPOLATE,E2 #INTERPOLATE,E3 #INTERPOLATE,E4 #INTERPOLATE,E5 #INTERPOLATE,E6 #INTERPOLATE}}}
DECL E6POS XIMM_PlaceApprPushUp={X 97.6707687,Y 58.7011833,Z 239.215240,A 90.0060806,B 1.10676742,C 0.0136310924,S 2,T 35,E1 0.0,E2 0.0,E3 0.0,E4 0.0,E5 0.0,E6 0.0}
DECL FDAT FIMM_PlaceApprPushUp={TOOL_NO 2,BASE_NO 3,IPO_FRAME #BASE,POINT2[] " "}
DECL LDAT LCPDAT12={VEL 0.100000,ACC 60.0000,APO_DIST 500.000,APO_FAC 50.0000,AXIS_VEL 100.000,AXIS_ACC 60.0000,ORI_TYP #VAR,CIRC_TYP #BASE,JERK_FAC 50.0000,GEAR_JERK 100.000,EXAX_IGN 0,CB {AUX_PT {ORI #CONSIDER,E1 #CONSIDER,E2 #CONSIDER,E3 #CONSIDER,E4 #CONSIDER,E5 #CONSIDER,E6 #CONSIDER},TARGET_PT {ORI #INTERPOLATE,E1 #INTERPOLATE,E2 #INTERPOLATE,E3 #INTERPOLATE,E4 #INTERPOLATE,E5 #INTERPOLATE,E6 #INTERPOLATE}}}
DECL LDAT LCPDAT13={VEL 0.100000,ACC 60.0000,APO_DIST 500.000,APO_FAC 50.0000,AXIS_VEL 100.000,AXIS_ACC 60.0000,ORI_TYP #VAR,CIRC_TYP #BASE,JERK_FAC 50.0000,GEAR_JERK 100.000,EXAX_IGN 0,CB {AUX_PT {ORI #CONSIDER,E1 #CONSIDER,E2 #CONSIDER,E3 #CONSIDER,E4 #CONSIDER,E5 #CONSIDER,E6 #CONSIDER},TARGET_PT {ORI #INTERPOLATE,E1 #INTERPOLATE,E2 #INTERPOLATE,E3 #INTERPOLATE,E4 #INTERPOLATE,E5 #INTERPOLATE,E6 #INTERPOLATE}}}
DECL LDAT LCPDAT14={VEL 1.00000,ACC 60.0000,APO_DIST 500.000,APO_FAC 50.0000,AXIS_VEL 100.000,AXIS_ACC 60.0000,ORI_TYP #VAR,CIRC_TYP #BASE,JERK_FAC 50.0000,GEAR_JERK 100.000,EXAX_IGN 0,CB {AUX_PT {ORI #CONSIDER,E1 #CONSIDER,E2 #CONSIDER,E3 #CONSIDER,E4 #CONSIDER,E5 #CONSIDER,E6 #CONSIDER},TARGET_PT {ORI #INTERPOLATE,E1 #INTERPOLATE,E2 #INTERPOLATE,E3 #INTERPOLATE,E4 #INTERPOLATE,E5 #INTERPOLATE,E6 #INTERPOLATE}}}
DECL E6POS XIMM_PlaceApprClose3={X 97.6714,Y 58.0502853,Z 241.592743,A 90.0060806,B 1.10676742,C 0.0136310868,S 2,T 35,E1 0.0,E2 0.0,E3 0.0,E4 0.0,E5 0.0,E6 0.0}
DECL FDAT FIMM_PlaceApprClose3={TOOL_NO 2,BASE_NO 3,IPO_FRAME #BASE,POINT2[] " "}
DECL LDAT LCPDAT15={VEL 0.100000,ACC 60.0000,APO_DIST 500.000,APO_FAC 50.0000,AXIS_VEL 100.000,AXIS_ACC 60.0000,ORI_TYP #VAR,CIRC_TYP #BASE,JERK_FAC 50.0000,GEAR_JERK 100.000,EXAX_IGN 0,CB {AUX_PT {ORI #CONSIDER,E1 #CONSIDER,E2 #CONSIDER,E3 #CONSIDER,E4 #CONSIDER,E5 #CONSIDER,E6 #CONSIDER},TARGET_PT {ORI #INTERPOLATE,E1 #INTERPOLATE,E2 #INTERPOLATE,E3 #INTERPOLATE,E4 #INTERPOLATE,E5 #INTERPOLATE,E6 #INTERPOLATE}}}
DECL LDAT LCPDAT16={VEL 0.100000,ACC 60.0000,APO_DIST 500.000,APO_FAC 50.0000,AXIS_VEL 100.000,AXIS_ACC 60.0000,ORI_TYP #VAR,CIRC_TYP #BASE,JERK_FAC 50.0000,GEAR_JERK 100.000,EXAX_IGN 0,CB {AUX_PT {ORI #CONSIDER,E1 #CONSIDER,E2 #CONSIDER,E3 #CONSIDER,E4 #CONSIDER,E5 #CONSIDER,E6 #CONSIDER},TARGET_PT {ORI #INTERPOLATE,E1 #INTERPOLATE,E2 #INTERPOLATE,E3 #INTERPOLATE,E4 #INTERPOLATE,E5 #INTERPOLATE,E6 #INTERPOLATE}}}
DECL LDAT LCPDAT17={VEL 0.0500000,ACC 60.0000,APO_DIST 500.000,APO_FAC 50.0000,AXIS_VEL 100.000,AXIS_ACC 60.0000,ORI_TYP #VAR,CIRC_TYP #BASE,JERK_FAC 50.0000,GEAR_JERK 100.000,EXAX_IGN 0,CB {AUX_PT {ORI #CONSIDER,E1 #CONSIDER,E2 #CONSIDER,E3 #CONSIDER,E4 #CONSIDER,E5 #CONSIDER,E6 #CONSIDER},TARGET_PT {ORI #INTERPOLATE,E1 #INTERPOLATE,E2 #INTERPOLATE,E3 #INTERPOLATE,E4 #INTERPOLATE,E5 #INTERPOLATE,E6 #INTERPOLATE}}}
DECL LDAT LCPDAT8={VEL 2.00000,ACC 60.0000,APO_DIST 500.000,APO_FAC 50.0000,AXIS_VEL 100.000,AXIS_ACC 60.0000,ORI_TYP #VAR,CIRC_TYP #BASE,JERK_FAC 50.0000,GEAR_JERK 100.000,EXAX_IGN 0,CB {AUX_PT {ORI #CONSIDER,E1 #CONSIDER,E2 #CONSIDER,E3 #CONSIDER,E4 #CONSIDER,E5 #CONSIDER,E6 #CONSIDER},TARGET_PT {ORI #INTERPOLATE,E1 #INTERPOLATE,E2 #INTERPOLATE,E3 #INTERPOLATE,E4 #INTERPOLATE,E5 #INTERPOLATE,E6 #INTERPOLATE}}}
DECL PDAT PPDAT12={VEL 100.000,ACC 60.0000,APO_DIST 500.000,APO_MODE #CDIS,GEAR_JERK 100.000,EXAX_IGN 0}
DECL PDAT PPDAT13={VEL 100.000,ACC 60.0000,APO_DIST 500.000,APO_MODE #CDIS,GEAR_JERK 100.000,EXAX_IGN 0}
DECL E6POS XIMM_PlaceSideShft1={X 98.1707687,Y 58.7012329,Z 239.215118,A 90.0060806,B 1.10676742,C 0.0136310877,S 2,T 35,E1 0.0,E2 0.0,E3 0.0,E4 0.0,E5 0.0,E6 0.0}
DECL FDAT FIMM_PlaceSideShft1={TOOL_NO 2,BASE_NO 3,IPO_FRAME #BASE,POINT2[] " "}
DECL LDAT LCPDAT18={VEL 2.00000,ACC 60.0000,APO_DIST 500.000,APO_FAC 50.0000,AXIS_VEL 100.000,AXIS_ACC 60.0000,ORI_TYP #VAR,CIRC_TYP #BASE,JERK_FAC 50.0000,GEAR_JERK 100.000,EXAX_IGN 0,CB {AUX_PT {ORI #CONSIDER,E1 #CONSIDER,E2 #CONSIDER,E3 #CONSIDER,E4 #CONSIDER,E5 #CONSIDER,E6 #CONSIDER},TARGET_PT {ORI #INTERPOLATE,E1 #INTERPOLATE,E2 #INTERPOLATE,E3 #INTERPOLATE,E4 #INTERPOLATE,E5 #INTERPOLATE,E6 #INTERPOLATE}}}
DECL E6POS XIMM_PlaceSideShft2={X 97.1707687,Y 58.7011337,Z 239.215363,A 90.0060806,B 1.10676742,C 0.0136310831,S 2,T 35,E1 0.0,E2 0.0,E3 0.0,E4 0.0,E5 0.0,E6 0.0}
DECL FDAT FIMM_PlaceSideShft2={TOOL_NO 2,BASE_NO 3,IPO_FRAME #BASE,POINT2[] " "}
DECL LDAT LCPDAT19={VEL 2.00000,ACC 60.0000,APO_DIST 500.000,APO_FAC 50.0000,AXIS_VEL 100.000,AXIS_ACC 60.0000,ORI_TYP #VAR,CIRC_TYP #BASE,JERK_FAC 50.0000,GEAR_JERK 100.000,EXAX_IGN 0,CB {AUX_PT {ORI #CONSIDER,E1 #CONSIDER,E2 #CONSIDER,E3 #CONSIDER,E4 #CONSIDER,E5 #CONSIDER,E6 #CONSIDER},TARGET_PT {ORI #INTERPOLATE,E1 #INTERPOLATE,E2 #INTERPOLATE,E3 #INTERPOLATE,E4 #INTERPOLATE,E5 #INTERPOLATE,E6 #INTERPOLATE}}}
DECL E6POS XIMM_PlaceSideShft3={X 97.6707687,Y 58.7011833,Z 239.215240,A 90.0060806,B 1.10676742,C 0.0136310924,S 2,T 35,E1 0.0,E2 0.0,E3 0.0,E4 0.0,E5 0.0,E6 0.0}
DECL FDAT FIMM_PlaceSideShft3={TOOL_NO 2,BASE_NO 3,IPO_FRAME #BASE,POINT2[] " "}
DECL LDAT LCPDAT20={VEL 2.00000,ACC 60.0000,APO_DIST 500.000,APO_FAC 50.0000,AXIS_VEL 100.000,AXIS_ACC 60.0000,ORI_TYP #VAR,CIRC_TYP #BASE,JERK_FAC 50.0000,GEAR_JERK 100.000,EXAX_IGN 0,CB {AUX_PT {ORI #CONSIDER,E1 #CONSIDER,E2 #CONSIDER,E3 #CONSIDER,E4 #CONSIDER,E5 #CONSIDER,E6 #CONSIDER},TARGET_PT {ORI #INTERPOLATE,E1 #INTERPOLATE,E2 #INTERPOLATE,E3 #INTERPOLATE,E4 #INTERPOLATE,E5 #INTERPOLATE,E6 #INTERPOLATE}}}
DECL LDAT LCPDAT21={VEL 0.0500000,ACC 60.0000,APO_DIST 500.000,APO_FAC 50.0000,AXIS_VEL 100.000,AXIS_ACC 60.0000,ORI_TYP #VAR,CIRC_TYP #BASE,JERK_FAC 50.0000,GEAR_JERK 100.000,EXAX_IGN 0,CB {AUX_PT {ORI #CONSIDER,E1 #CONSIDER,E2 #CONSIDER,E3 #CONSIDER,E4 #CONSIDER,E5 #CONSIDER,E6 #CONSIDER},TARGET_PT {ORI #INTERPOLATE,E1 #INTERPOLATE,E2 #INTERPOLATE,E3 #INTERPOLATE,E4 #INTERPOLATE,E5 #INTERPOLATE,E6 #INTERPOLATE}}}
DECL PDAT PPDAT14={VEL 100.000,ACC 60.0000,APO_DIST 500.000,APO_MODE #CDIS,GEAR_JERK 100.000,EXAX_IGN 0}
DECL LDAT LCPDAT22={VEL 2.00000,ACC 60.0000,APO_DIST 500.000,APO_FAC 50.0000,AXIS_VEL 100.000,AXIS_ACC 60.0000,ORI_TYP #VAR,CIRC_TYP #BASE,JERK_FAC 50.0000,GEAR_JERK 100.000,EXAX_IGN 0,CB {AUX_PT {ORI #CONSIDER,E1 #CONSIDER,E2 #CONSIDER,E3 #CONSIDER,E4 #CONSIDER,E5 #CONSIDER,E6 #CONSIDER},TARGET_PT {ORI #INTERPOLATE,E1 #INTERPOLATE,E2 #INTERPOLATE,E3 #INTERPOLATE,E4 #INTERPOLATE,E5 #INTERPOLATE,E6 #INTERPOLATE}}}
DECL PDAT PPDAT15={VEL 100.000,ACC 60.0000,APO_DIST 500.000,APO_MODE #CDIS,GEAR_JERK 100.000,EXAX_IGN 0}
DECL LDAT LCPDAT28={VEL 0.500000,ACC 60.0000,APO_DIST 500.000,APO_FAC 50.0000,AXIS_VEL 100.000,AXIS_ACC 60.0000,ORI_TYP #VAR,CIRC_TYP #BASE,JERK_FAC 50.0000,GEAR_JERK 100.000,EXAX_IGN 0,CB {AUX_PT {ORI #CONSIDER,E1 #CONSIDER,E2 #CONSIDER,E3 #CONSIDER,E4 #CONSIDER,E5 #CONSIDER,E6 #CONSIDER},TARGET_PT {ORI #INTERPOLATE,E1 #INTERPOLATE,E2 #INTERPOLATE,E3 #INTERPOLATE,E4 #INTERPOLATE,E5 #INTERPOLATE,E6 #INTERPOLATE}}}
DECL LDAT LCPDAT29={VEL 2.00000,ACC 60.0000,APO_DIST 500.000,APO_FAC 50.0000,AXIS_VEL 100.000,AXIS_ACC 60.0000,ORI_TYP #VAR,CIRC_TYP #BASE,JERK_FAC 50.0000,GEAR_JERK 100.000,EXAX_IGN 0,CB {AUX_PT {ORI #CONSIDER,E1 #CONSIDER,E2 #CONSIDER,E3 #CONSIDER,E4 #CONSIDER,E5 #CONSIDER,E6 #CONSIDER},TARGET_PT {ORI #INTERPOLATE,E1 #INTERPOLATE,E2 #INTERPOLATE,E3 #INTERPOLATE,E4 #INTERPOLATE,E5 #INTERPOLATE,E6 #INTERPOLATE}}}
DECL E6POS XIMM_PickApprFault={X 94.9665527,Y 11.0926991,Z 52.7965889,A -90.3063202,B -1.35644329,C -177.577133,S 2,T 35,E1 0.0,E2 0.0,E3 0.0,E4 0.0,E5 0.0,E6 0.0}
DECL FDAT FIMM_PickApprFault={TOOL_NO 2,BASE_NO 3,IPO_FRAME #BASE,POINT2[] " "}
DECL LDAT LCPDAT30={VEL 2.00000,ACC 60.0000,APO_DIST 500.000,APO_FAC 50.0000,AXIS_VEL 100.000,AXIS_ACC 60.0000,ORI_TYP #VAR,CIRC_TYP #BASE,JERK_FAC 50.0000,GEAR_JERK 100.000,EXAX_IGN 0,CB {AUX_PT {ORI #CONSIDER,E1 #CONSIDER,E2 #CONSIDER,E3 #CONSIDER,E4 #CONSIDER,E5 #CONSIDER,E6 #CONSIDER},TARGET_PT {ORI #INTERPOLATE,E1 #INTERPOLATE,E2 #INTERPOLATE,E3 #INTERPOLATE,E4 #INTERPOLATE,E5 #INTERPOLATE,E6 #INTERPOLATE}}}
DECL LDAT LCPDAT31={VEL 0.500000,ACC 60.0000,APO_DIST 500.000,APO_FAC 50.0000,AXIS_VEL 100.000,AXIS_ACC 60.0000,ORI_TYP #VAR,CIRC_TYP #BASE,JERK_FAC 50.0000,GEAR_JERK 100.000,EXAX_IGN 0,CB {AUX_PT {ORI #CONSIDER,E1 #CONSIDER,E2 #CONSIDER,E3 #CONSIDER,E4 #CONSIDER,E5 #CONSIDER,E6 #CONSIDER},TARGET_PT {ORI #INTERPOLATE,E1 #INTERPOLATE,E2 #INTERPOLATE,E3 #INTERPOLATE,E4 #INTERPOLATE,E5 #INTERPOLATE,E6 #INTERPOLATE}}}
DECL E6POS XIMM_PickApprFault2={X 94.7874,Y 71.5678711,Z 51.3433838,A -90.3063202,B -1.35644329,C -177.577133,S 2,T 35,E1 0.0,E2 0.0,E3 0.0,E4 0.0,E5 0.0,E6 0.0}
DECL FDAT FIMM_PickApprFault2={TOOL_NO 2,BASE_NO 3,IPO_FRAME #BASE,POINT2[] " "}
DECL LDAT LCPDAT32={VEL 0.500000,ACC 60.0000,APO_DIST 500.000,APO_FAC 50.0000,AXIS_VEL 100.000,AXIS_ACC 60.0000,ORI_TYP #VAR,CIRC_TYP #BASE,JERK_FAC 50.0000,GEAR_JERK 100.000,EXAX_IGN 0,CB {AUX_PT {ORI #CONSIDER,E1 #CONSIDER,E2 #CONSIDER,E3 #CONSIDER,E4 #CONSIDER,E5 #CONSIDER,E6 #CONSIDER},TARGET_PT {ORI #INTERPOLATE,E1 #INTERPOLATE,E2 #INTERPOLATE,E3 #INTERPOLATE,E4 #INTERPOLATE,E5 #INTERPOLATE,E6 #INTERPOLATE}}}
DECL LDAT LCPDAT9={VEL 2.00000,ACC 60.0000,APO_DIST 500.000,APO_FAC 50.0000,AXIS_VEL 100.000,AXIS_ACC 60.0000,ORI_TYP #VAR,CIRC_TYP #BASE,JERK_FAC 50.0000,GEAR_JERK 100.000,EXAX_IGN 0,CB {AUX_PT {ORI #CONSIDER,E1 #CONSIDER,E2 #CONSIDER,E3 #CONSIDER,E4 #CONSIDER,E5 #CONSIDER,E6 #CONSIDER},TARGET_PT {ORI #INTERPOLATE,E1 #INTERPOLATE,E2 #INTERPOLATE,E3 #INTERPOLATE,E4 #INTERPOLATE,E5 #INTERPOLATE,E6 #INTERPOLATE}}}
DECL LDAT LCPDAT23={VEL 2.00000,ACC 60.0000,APO_DIST 500.000,APO_FAC 50.0000,AXIS_VEL 100.000,AXIS_ACC 60.0000,ORI_TYP #VAR,CIRC_TYP #BASE,JERK_FAC 50.0000,GEAR_JERK 100.000,EXAX_IGN 0,CB {AUX_PT {ORI #CONSIDER,E1 #CONSIDER,E2 #CONSIDER,E3 #CONSIDER,E4 #CONSIDER,E5 #CONSIDER,E6 #CONSIDER},TARGET_PT {ORI #INTERPOLATE,E1 #INTERPOLATE,E2 #INTERPOLATE,E3 #INTERPOLATE,E4 #INTERPOLATE,E5 #INTERPOLATE,E6 #INTERPOLATE}}}
DECL LDAT LCPDAT24={VEL 2.00000,ACC 100.000,APO_DIST 500.000,APO_FAC 50.0000,AXIS_VEL 100.000,AXIS_ACC 100.000,ORI_TYP #VAR,CIRC_TYP #BASE,JERK_FAC 50.0000,GEAR_JERK 100.000,EXAX_IGN 0,CB {AUX_PT {ORI #CONSIDER,E1 #CONSIDER,E2 #CONSIDER,E3 #CONSIDER,E4 #CONSIDER,E5 #CONSIDER,E6 #CONSIDER},TARGET_PT {ORI #INTERPOLATE,E1 #INTERPOLATE,E2 #INTERPOLATE,E3 #INTERPOLATE,E4 #INTERPOLATE,E5 #INTERPOLATE,E6 #INTERPOLATE}}}
DECL E6POS XIMM_PlaceSideShft4={X 98.1707687,Y 58.7012329,Z 239.215118,A 90.0060806,B 1.10676742,C 0.0136310877,S 2,T 35,E1 0.0,E2 0.0,E3 0.0,E4 0.0,E5 0.0,E6 0.0}
DECL FDAT FIMM_PlaceSideShft4={TOOL_NO 2,BASE_NO 3,IPO_FRAME #BASE,POINT2[] " "}
DECL LDAT LCPDAT25={VEL 2.00000,ACC 60.0000,APO_DIST 500.000,APO_FAC 50.0000,AXIS_VEL 100.000,AXIS_ACC 60.0000,ORI_TYP #VAR,CIRC_TYP #BASE,JERK_FAC 50.0000,GEAR_JERK 100.000,EXAX_IGN 0,CB {AUX_PT {ORI #CONSIDER,E1 #CONSIDER,E2 #CONSIDER,E3 #CONSIDER,E4 #CONSIDER,E5 #CONSIDER,E6 #CONSIDER},TARGET_PT {ORI #INTERPOLATE,E1 #INTERPOLATE,E2 #INTERPOLATE,E3 #INTERPOLATE,E4 #INTERPOLATE,E5 #INTERPOLATE,E6 #INTERPOLATE}}}
ENDDAT
